LIN {X 0,Y 310.656,Z 1014.601,A -85,B 0,C 180,E1 26309.689,E2 26309.689} C_VEL
LIN {X 0,Y 289.727,Z 1045.579,A -85,B 0,C 180,E1 26313.885,E2 26313.885} C_VEL
LIN {X 0,Y 277.793,Z 1061.064,A -85,B 0,C 180,E1 26316.691,E2 26316.691} C_VEL
LIN {X 0,Y 266.703,Z 1071.977,A -85,B 0,C 180,E1 26318.403,E2 26318.403} C_VEL
LIN {X 0,Y 255.321,Z 1081.969,A -85,B 0,C 180,E1 26320.351,E2 26320.351} C_VEL
LIN {X 0,Y 233.204,Z 1105.025,A -85,B 0,C 180,E1 26328.775,E2 26328.775} C_VEL
LIN {X 0,Y 215.813,Z 1122.452,A -85,B 0,C 180,E1 26339.407,E2 26339.407} C_VEL
LIN {X 0,Y 205.814,Z 1133.022,A -85,B 0,C 180,E1 26350.657,E2 26350.657} C_VEL
LIN {X 0,Y 201.917,Z 1138.235,A -85,B 0,C 180,E1 26361.372,E2 26361.372} C_VEL
LIN {X 0,Y 201.653,Z 1139.483,A -85,B 0,C 180,E1 26370.004,E2 26370.004} C_VEL
LIN {X 0,Y 201.955,Z 1138.196,A -85,B 0,C 180,E1 26378.634,E2 26378.634} C_VEL
LIN {X 0,Y 205.859,Z 1132.908,A -85,B 0,C 180,E1 26389.346,E2 26389.346} C_VEL
LIN {X 0,Y 215.912,Z 1122.258,A -85,B 0,C 180,E1 26400.586,E2 26400.586} C_VEL
LIN {X 0,Y 233.437,Z 1104.704,A -85,B 0,C 180,E1 26411.215,E2 26411.215} C_VEL
LIN {X 0,Y 255.523,Z 1081.509,A -85,B 0,C 180,E1 26419.657,E2 26419.657} C_VEL
LIN {X 0,Y 278.933,Z 1053.943,A -85,B 0,C 180,E1 26425.937,E2 26425.937} C_VEL
LIN {X 0,Y 303.43,Z 1019.934,A -85,B 0,C 180,E1 26430.914,E2 26430.914} C_VEL
LIN {X 0,Y 325.476,Z 982.197,A -85,B 0,C 180,E1 26434.492,E2 26434.492} C_VEL
LIN {X 0,Y 325.74,Z 970.343,A -85,B 0,C 180,E1 26437.786,E2 26437.786} C_VEL
LIN {X 0,Y 324.423,Z 954.359,A -85,B 0,C 180,E1 26443.718,E2 26443.718} C_VEL
LIN {X 0,Y 322.918,Z 944.433,A -85,B 0,C 180,E1 26449.173,E2 26449.173} C_VEL
LIN {X 0,Y 322.497,Z 936.41,A -85,B 0,C 180,E1 26457.297,E2 26457.297} C_VEL
LIN {X 0,Y 322.512,Z 936.483,A -85,B 0,C 180,E1 26459.99,E2 26459.99} C_VEL
LIN {X 0,Y 322.75,Z 943.035,A -85,B 0,C 180,E1 26466.729,E2 26466.729} C_VEL
LIN {X 0,Y 324.195,Z 953.745,A -85,B 0,C 180,E1 26472.815,E2 26472.815} C_VEL
LIN {X 0,Y 325.518,Z 969.409,A -85,B 0,C 180,E1 26478.651,E2 26478.651} C_VEL
LIN {X 0,Y 325.37,Z 982.593,A -85,B 0,C 180,E1 26482.362,E2 26482.362} C_VEL
LIN {X 0,Y 303.394,Z 1021.107,A -85,B 0,C 180,E1 26485.977,E2 26485.977} C_VEL
LIN {X 0,Y 280.23,Z 1054.421,A -85,B 0,C 180,E1 26490.68,E2 26490.68} C_VEL
LIN {X 0,Y 257.476,Z 1082.65,A -85,B 0,C 180,E1 26496.694,E2 26496.694} C_VEL
LIN {X 0,Y 237.226,Z 1105.526,A -85,B 0,C 180,E1 26504.062,E2 26504.062} C_VEL
LIN {X 0,Y 219.041,Z 1125.176,A -85,B 0,C 180,E1 26513.983,E2 26513.983} C_VEL
LIN {X 0,Y 206.829,Z 1139.423,A -85,B 0,C 180,E1 26525.882,E2 26525.882} C_VEL
LIN {X 0,Y 202.177,Z 1146.947,A -85,B 0,C 180,E1 26537.003,E2 26537.003} C_VEL
LIN {X 0,Y 201.199,Z 1149.691,A -85,B 0,C 180,E1 26545.677,E2 26545.677} C_VEL
LIN {X 0,Y 201.527,Z 1150.057,A -85,B 0,C 180,E1 26549.996,E2 26549.996} C_VEL
LIN {X 0,Y 201.398,Z 1148.668,A -85,B 0,C 180,E1 26558.65,E2 26558.65} C_VEL
LIN {X 0,Y 204.311,Z 1143.178,A -85,B 0,C 180,E1 26569.491,E2 26569.491} C_VEL
LIN {X 0,Y 213.682,Z 1131.328,A -85,B 0,C 180,E1 26581.729,E2 26581.729} C_VEL
LIN {X 0,Y 229.673,Z 1113.75,A -85,B 0,C 180,E1 26592.392,E2 26592.392} C_VEL
LIN {X 0,Y 250.76,Z 1090.55,A -85,B 0,C 180,E1 26601.146,E2 26601.146} C_VEL
LIN {X 0,Y 272.752,Z 1064.306,A -85,B 0,C 180,E1 26607.53,E2 26607.53} C_VEL
LIN {X 0,Y 295.471,Z 1033.482,A -85,B 0,C 180,E1 26612.53,E2 26612.53} C_VEL
LIN {X 0,Y 318.003,Z 997.074,A -85,B 0,C 180,E1 26616.452,E2 26616.452} C_VEL
LIN {X 0,Y 325.814,Z 981.719,A -85,B 0,C 180,E1 26617.813,E2 26617.813} C_VEL
LIN {X 0,Y 325.351,Z 964.308,A -85,B 0,C 180,E1 26623.09,E2 26623.09} C_VEL
LIN {X 0,Y 324,Z 951.083,A -85,B 0,C 180,E1 26628.548,E2 26628.548} C_VEL
LIN {X 0,Y 322.759,Z 941.668,A -85,B 0,C 180,E1 26634.623,E2 26634.623} C_VEL
LIN {X 0,Y 322.742,Z 936.78,A -85,B 0,C 180,E1 26640.01,E2 26640.01} C_VEL
LIN {X 0,Y 322.687,Z 936.823,A -85,B 0,C 180,E1 26642.701,E2 26642.701} C_VEL
LIN {X 0,Y 323.156,Z 944.767,A -85,B 0,C 180,E1 26650.819,E2 26650.819} C_VEL
LIN {X 0,Y 324.807,Z 956.324,A -85,B 0,C 180,E1 26656.96,E2 26656.96} C_VEL
LIN {X 0,Y 326.013,Z 972.408,A -85,B 0,C 180,E1 26662.739,E2 26662.739} C_VEL
LIN {X 0,Y 326.137,Z 981.075,A -85,B 0,C 180,E1 26665.251,E2 26665.251} C_VEL
LIN {X 0,Y 303.951,Z 1019.446,A -85,B 0,C 180,E1 26668.904,E2 26668.904} C_VEL
LIN {X 0,Y 280.08,Z 1052.757,A -85,B 0,C 180,E1 26673.726,E2 26673.726} C_VEL
LIN {X 0,Y 255.321,Z 1081.969,A -85,B 0,C 180,E1 26680.351,E2 26680.351} C_VEL
LIN {X 0,Y 243.945,Z 1091.297,A -85,B 0,C 180,E1 26682.559,E2 26682.559} C_VEL
LIN {X 0,Y 232.748,Z 1099.829,A -85,B 0,C 180,E1 26685.058,E2 26685.058} C_VEL
LIN {X 0,Y 214.056,Z 1117.775,A -85,B 0,C 180,E1 26694.59,E2 26694.59} C_VEL
LIN {X 0,Y 201.342,Z 1130.014,A -85,B 0,C 180,E1 26705.583,E2 26705.583} C_VEL
LIN {X 0,Y 195.265,Z 1136.858,A -85,B 0,C 180,E1 26716.543,E2 26716.543} C_VEL
LIN {X 0,Y 193.614,Z 1139.385,A -85,B 0,C 180,E1 26725.516,E2 26725.516} C_VEL
LIN {X 0,Y 193.779,Z 1139.69,A -85,B 0,C 180,E1 26730.004,E2 26730.004} C_VEL
LIN {X 0,Y 194.118,Z 1138.404,A -85,B 0,C 180,E1 26738.985,E2 26738.985} C_VEL
LIN {X 0,Y 198.32,Z 1133.12,A -85,B 0,C 180,E1 26750.113,E2 26750.113} C_VEL
LIN {X 0,Y 209.02,Z 1122.475,A -85,B 0,C 180,E1 26761.709,E2 26761.709} C_VEL
LIN {X 0,Y 227.721,Z 1104.651,A -85,B 0,C 180,E1 26772.674,E2 26772.674} C_VEL
LIN {X 0,Y 250.602,Z 1081.533,A -85,B 0,C 180,E1 26781.113,E2 26781.113} C_VEL
LIN {X 0,Y 275.896,Z 1052.531,A -85,B 0,C 180,E1 26787.609,E2 26787.609} C_VEL
LIN {X 0,Y 300.384,Z 1019.113,A -85,B 0,C 180,E1 26792.364,E2 26792.364} C_VEL
LIN {X 0,Y 320.943,Z 984.275,A -85,B 0,C 180,E1 26795.727,E2 26795.727} C_VEL
LIN {X 0,Y 320.748,Z 967.42,A -85,B 0,C 180,E1 26801.325,E2 26801.325} C_VEL
LIN {X 0,Y 319.765,Z 955.09,A -85,B 0,C 180,E1 26806.984,E2 26806.984} C_VEL
LIN {X 0,Y 318.752,Z 947.169,A -85,B 0,C 180,E1 26813.041,E2 26813.041} C_VEL
LIN {X 0,Y 319.14,Z 943.671,A -85,B 0,C 180,E1 26817.269,E2 26817.269} C_VEL
LIN {X 0,Y 319.16,Z 943.724,A -85,B 0,C 180,E1 26819.99,E2 26819.99} C_VEL
LIN {X 0,Y 319.148,Z 950.325,A -85,B 0,C 180,E1 26826.806,E2 26826.806} C_VEL
LIN {X 0,Y 320.193,Z 961.352,A -85,B 0,C 180,E1 26832.978,E2 26832.978} C_VEL
LIN {X 0,Y 320.821,Z 974.906,A -85,B 0,C 180,E1 26838.092,E2 26838.092} C_VEL
LIN {X 0,Y 320.66,Z 985.105,A -85,B 0,C 180,E1 26841.15,E2 26841.15} C_VEL
LIN {X 0,Y 297.827,Z 1024.077,A -85,B 0,C 180,E1 26844.959,E2 26844.959} C_VEL
LIN {X 0,Y 272.881,Z 1058.44,A -85,B 0,C 180,E1 26849.965,E2 26849.965} C_VEL
LIN {X 0,Y 247.91,Z 1087.811,A -85,B 0,C 180,E1 26856.658,E2 26856.658} C_VEL
LIN {X 0,Y 225.003,Z 1112.055,A -85,B 0,C 180,E1 26865.528,E2 26865.528} C_VEL
LIN {X 0,Y 208.116,Z 1129.468,A -85,B 0,C 180,E1 26875.905,E2 26875.905} C_VEL
LIN {X 0,Y 197.83,Z 1141.286,A -85,B 0,C 180,E1 26887.48,E2 26887.48} C_VEL
LIN {X 0,Y 194.384,Z 1146.736,A -85,B 0,C 180,E1 26896.473,E2 26896.473} C_VEL
LIN {X 0,Y 193.286,Z 1149.483,A -85,B 0,C 180,E1 26905.5,E2 26905.5} C_VEL
LIN {X 0,Y 193.627,Z 1149.85,A -85,B 0,C 180,E1 26909.996,E2 26909.996} C_VEL
LIN {X 0,Y 193.516,Z 1148.459,A -85,B 0,C 180,E1 26919.005,E2 26919.005} C_VEL
LIN {X 0,Y 196.695,Z 1142.965,A -85,B 0,C 180,E1 26930.278,E2 26930.278} C_VEL
LIN {X 0,Y 206.766,Z 1131.11,A -85,B 0,C 180,E1 26942.922,E2 26942.922} C_VEL
LIN {X 0,Y 225.038,Z 1112.176,A -85,B 0,C 180,E1 26954.462,E2 26954.462} C_VEL
LIN {X 0,Y 247.896,Z 1087.996,A -85,B 0,C 180,E1 26963.337,E2 26963.337} C_VEL
LIN {X 0,Y 272.926,Z 1058.613,A -85,B 0,C 180,E1 26970.041,E2 26970.041} C_VEL
LIN {X 0,Y 297.899,Z 1024.305,A -85,B 0,C 180,E1 26975.04,E2 26975.04} C_VEL
LIN {X 0,Y 320.005,Z 987.274,A -85,B 0,C 180,E1 26978.578,E2 26978.578} C_VEL
LIN {X 0,Y 320.914,Z 984.537,A -85,B 0,C 180,E1 26979.05,E2 26979.05} C_VEL
LIN {X 0,Y 320.856,Z 968.383,A -85,B 0,C 180,E1 26984.257,E2 26984.257} C_VEL
LIN {X 0,Y 319.943,Z 956.175,A -85,B 0,C 180,E1 26989.712,E2 26989.712} C_VEL
LIN {X 0,Y 319.033,Z 947.677,A -85,B 0,C 180,E1 26995.786,E2 26995.786} C_VEL
LIN {X 0,Y 319.368,Z 944.031,A -85,B 0,C 180,E1 27000.01,E2 27000.01} C_VEL
LIN {X 0,Y 319.294,Z 944.109,A -85,B 0,C 180,E1 27002.73,E2 27002.73} C_VEL
LIN {X 0,Y 319.368,Z 950.839,A -85,B 0,C 180,E1 27009.986,E2 27009.986} C_VEL
LIN {X 0,Y 320.468,Z 960.823,A -85,B 0,C 180,E1 27015.784,E2 27015.784} C_VEL
LIN {X 0,Y 321.21,Z 976.997,A -85,B 0,C 180,E1 27021.908,E2 27021.908} C_VEL
LIN {X 0,Y 320.622,Z 985.751,A -85,B 0,C 180,E1 27024.382,E2 27024.382} C_VEL
LIN {X 0,Y 299.451,Z 1020.785,A -85,B 0,C 180,E1 27027.697,E2 27027.697} C_VEL
LIN {X 0,Y 275.707,Z 1053.01,A -85,B 0,C 180,E1 27032.34,E2 27032.34} C_VEL
LIN {X 0,Y 250.422,Z 1081.958,A -85,B 0,C 180,E1 27038.881,E2 27038.881} C_VEL
LIN {X 0,Y 232.748,Z 1099.829,A -85,B 0,C 180,E1 27045.058,E2 27045.058} C_VEL
LIN {X 0,Y 221.764,Z 1107.624,A -85,B 0,C 180,E1 27047.903,E2 27047.903} C_VEL
LIN {X 0,Y 211.211,Z 1114.605,A -85,B 0,C 180,E1 27051.106,E2 27051.106} C_VEL
LIN {X 0,Y 196.097,Z 1128.332,A -85,B 0,C 180,E1 27062.385,E2 27062.385} C_VEL
LIN {X 0,Y 187.522,Z 1137.066,A -85,B 0,C 180,E1 27075.976,E2 27075.976} C_VEL
LIN {X 0,Y 185.714,Z 1139.592,A -85,B 0,C 180,E1 27085.324,E2 27085.324} C_VEL
LIN {X 0,Y 185.873,Z 1139.897,A -85,B 0,C 180,E1 27090.004,E2 27090.004} C_VEL
LIN {X 0,Y 186.27,Z 1138.613,A -85,B 0,C 180,E1 27099.367,E2 27099.367} C_VEL
LIN {X 0,Y 190.839,Z 1133.33,A -85,B 0,C 180,E1 27110.937,E2 27110.937} C_VEL
LIN {X 0,Y 202.233,Z 1122.691,A -85,B 0,C 180,E1 27122.905,E2 27122.905} C_VEL
LIN {X 0,Y 221.862,Z 1104.875,A -85,B 0,C 180,E1 27134.085,E2 27134.085} C_VEL
LIN {X 0,Y 245.883,Z 1081.522,A -85,B 0,C 180,E1 27142.633,E2 27142.633} C_VEL
LIN {X 0,Y 271.691,Z 1052.79,A -85,B 0,C 180,E1 27149.035,E2 27149.035} C_VEL
LIN {X 0,Y 296.781,Z 1019.409,A -85,B 0,C 180,E1 27153.723,E2 27153.723} C_VEL
LIN {X 0,Y 315.966,Z 987.623,A -85,B 0,C 180,E1 27156.843,E2 27156.843} C_VEL
LIN {X 0,Y 316.206,Z 971.619,A -85,B 0,C 180,E1 27162.493,E2 27162.493} C_VEL
LIN {X 0,Y 315.6,Z 960.15,A -85,B 0,C 180,E1 27168.217,E2 27168.217} C_VEL
LIN {X 0,Y 315.145,Z 953.094,A -85,B 0,C 180,E1 27174.472,E2 27174.472} C_VEL
LIN {X 0,Y 315.586,Z 950.823,A -85,B 0,C 180,E1 27177.238,E2 27177.238} C_VEL
LIN {X 0,Y 315.604,Z 950.871,A -85,B 0,C 180,E1 27179.99,E2 27179.99} C_VEL
LIN {X 0,Y 315.429,Z 957.619,A -85,B 0,C 180,E1 27186.886,E2 27186.886} C_VEL
LIN {X 0,Y 315.999,Z 967.366,A -85,B 0,C 180,E1 27192.449,E2 27192.449} C_VEL
LIN {X 0,Y 316.083,Z 981.734,A -85,B 0,C 180,E1 27197.954,E2 27197.954} C_VEL
LIN {X 0,Y 315.726,Z 988.26,A -85,B 0,C 180,E1 27199.995,E2 27199.995} C_VEL
LIN {X 0,Y 311.446,Z 996.743,A -85,B 0,C 180,E1 27200.869,E2 27200.869} C_VEL
LIN {X 0,Y 286.904,Z 1034.674,A -85,B 0,C 180,E1 27204.854,E2 27204.854} C_VEL
LIN {X 0,Y 261.02,Z 1067.638,A -85,B 0,C 180,E1 27210.287,E2 27210.287} C_VEL
LIN {X 0,Y 236.125,Z 1094.834,A -85,B 0,C 180,E1 27217.354,E2 27217.354} C_VEL
LIN {X 0,Y 214.378,Z 1116.537,A -85,B 0,C 180,E1 27226.436,E2 27226.436} C_VEL
LIN {X 0,Y 197.865,Z 1132.819,A -85,B 0,C 180,E1 27237.582,E2 27237.582} C_VEL
LIN {X 0,Y 189.098,Z 1142.697,A -85,B 0,C 180,E1 27248.861,E2 27248.861} C_VEL
LIN {X 0,Y 185.658,Z 1148.233,A -85,B 0,C 180,E1 27260.602,E2 27260.602} C_VEL
LIN {X 0,Y 185.715,Z 1149.642,A -85,B 0,C 180,E1 27269.996,E2 27269.996} C_VEL
LIN {X 0,Y 186.127,Z 1147.185,A -85,B 0,C 180,E1 27282.456,E2 27282.456} C_VEL
LIN {X 0,Y 191.281,Z 1140.142,A -85,B 0,C 180,E1 27294.826,E2 27294.826} C_VEL
LIN {X 0,Y 204.521,Z 1126.321,A -85,B 0,C 180,E1 27307.66,E2 27307.66} C_VEL
LIN {X 0,Y 224.032,Z 1107.203,A -85,B 0,C 180,E1 27318.063,E2 27318.063} C_VEL
LIN {X 0,Y 247.226,Z 1083.229,A -85,B 0,C 180,E1 27326.108,E2 27326.108} C_VEL
LIN {X 0,Y 272.003,Z 1054.516,A -85,B 0,C 180,E1 27332.2,E2 27332.2} C_VEL
LIN {X 0,Y 296.648,Z 1020.872,A -85,B 0,C 180,E1 27336.827,E2 27336.827} C_VEL
LIN {X 0,Y 315.242,Z 990.373,A -85,B 0,C 180,E1 27339.661,E2 27339.661} C_VEL
LIN {X 0,Y 316.212,Z 983.473,A -85,B 0,C 180,E1 27341.563,E2 27341.563} C_VEL
LIN {X 0,Y 316.28,Z 969.136,A -85,B 0,C 180,E1 27346.859,E2 27346.859} C_VEL
LIN {X 0,Y 315.684,Z 959.928,A -85,B 0,C 180,E1 27351.732,E2 27351.732} C_VEL
LIN {X 0,Y 315.359,Z 953.613,A -85,B 0,C 180,E1 27357.257,E2 27357.257} C_VEL
LIN {X 0,Y 315.795,Z 951.212,A -85,B 0,C 180,E1 27360.01,E2 27360.01} C_VEL
LIN {X 0,Y 315.72,Z 951.302,A -85,B 0,C 180,E1 27362.761,E2 27362.761} C_VEL
LIN {X 0,Y 315.603,Z 957.552,A -85,B 0,C 180,E1 27369.683,E2 27369.683} C_VEL
LIN {X 0,Y 316.281,Z 966.936,A -85,B 0,C 180,E1 27375.287,E2 27375.287} C_VEL
LIN {X 0,Y 316.444,Z 982.685,A -85,B 0,C 180,E1 27381.422,E2 27381.422} C_VEL
LIN {X 0,Y 315.569,Z 989.407,A -85,B 0,C 180,E1 27383.343,E2 27383.343} C_VEL
LIN {X 0,Y 294.362,Z 1023.137,A -85,B 0,C 180,E1 27386.582,E2 27386.582} C_VEL
LIN {X 0,Y 270.127,Z 1054.868,A -85,B 0,C 180,E1 27391.203,E2 27391.203} C_VEL
LIN {X 0,Y 244.652,Z 1082.994,A -85,B 0,C 180,E1 27397.663,E2 27397.663} C_VEL
LIN {X 0,Y 221.552,Z 1105.307,A -85,B 0,C 180,E1 27405.966,E2 27405.966} C_VEL
LIN {X 0,Y 211.211,Z 1114.605,A -85,B 0,C 180,E1 27411.106,E2 27411.106} C_VEL
LIN {X 0,Y 201.172,Z 1120.795,A -85,B 0,C 180,E1 27414.718,E2 27414.718} C_VEL
LIN {X 0,Y 191.732,Z 1126.166,A -85,B 0,C 180,E1 27418.74,E2 27418.74} C_VEL
LIN {X 0,Y 181.895,Z 1135.042,A -85,B 0,C 180,E1 27430.542,E2 27430.542} C_VEL
LIN {X 0,Y 178.397,Z 1138.858,A -85,B 0,C 180,E1 27440.224,E2 27440.224} C_VEL
LIN {X 0,Y 177.967,Z 1140.104,A -85,B 0,C 180,E1 27450.004,E2 27450.004} C_VEL
LIN {X 0,Y 178.431,Z 1138.821,A -85,B 0,C 180,E1 27459.782,E2 27459.782} C_VEL
LIN {X 0,Y 183.396,Z 1133.542,A -85,B 0,C 180,E1 27471.83,E2 27471.83} C_VEL
LIN {X 0,Y 195.521,Z 1122.908,A -85,B 0,C 180,E1 27484.187,E2 27484.187} C_VEL
LIN {X 0,Y 215.598,Z 1105.61,A -85,B 0,C 180,E1 27495.334,E2 27495.334} C_VEL
LIN {X 0,Y 240.306,Z 1082.573,A -85,B 0,C 180,E1 27503.919,E2 27503.919} C_VEL
LIN {X 0,Y 267.655,Z 1053.048,A -85,B 0,C 180,E1 27510.506,E2 27510.506} C_VEL
LIN {X 0,Y 293.342,Z 1019.701,A -85,B 0,C 180,E1 27515.118,E2 27515.118} C_VEL
LIN {X 0,Y 311.02,Z 991.738,A -85,B 0,C 180,E1 27517.766,E2 27517.766} C_VEL
LIN {X 0,Y 311.679,Z 977.397,A -85,B 0,C 180,E1 27523.032,E2 27523.032} C_VEL
LIN {X 0,Y 311.561,Z 966.366,A -85,B 0,C 180,E1 27528.773,E2 27528.773} C_VEL
LIN {X 0,Y 311.557,Z 959.011,A -85,B 0,C 180,E1 27535.807,E2 27535.807} C_VEL
LIN {X 0,Y 311.897,Z 957.937,A -85,B 0,C 180,E1 27537.205,E2 27537.205} C_VEL
LIN {X 0,Y 311.923,Z 957.969,A -85,B 0,C 180,E1 27539.99,E2 27539.99} C_VEL
LIN {X 0,Y 311.516,Z 965.778,A -85,B 0,C 180,E1 27547.675,E2 27547.675} C_VEL
LIN {X 0,Y 311.614,Z 976.784,A -85,B 0,C 180,E1 27553.467,E2 27553.467} C_VEL
LIN {X 0,Y 310.921,Z 991.253,A -85,B 0,C 180,E1 27558.745,E2 27558.745} C_VEL
LIN {X 0,Y 310.239,Z 993.591,A -85,B 0,C 180,E1 27559.242,E2 27559.242} C_VEL
LIN {X 0,Y 287.46,Z 1028.955,A -85,B 0,C 180,E1 27562.714,E2 27562.714} C_VEL
LIN {X 0,Y 262.378,Z 1061.082,A -85,B 0,C 180,E1 27567.498,E2 27567.498} C_VEL
LIN {X 0,Y 237.267,Z 1088.591,A -85,B 0,C 180,E1 27573.879,E2 27573.879} C_VEL
LIN {X 0,Y 212.845,Z 1112.347,A -85,B 0,C 180,E1 27582.797,E2 27582.797} C_VEL
LIN {X 0,Y 193.685,Z 1130.122,A -85,B 0,C 180,E1 27594.071,E2 27594.071} C_VEL
LIN {X 0,Y 182.956,Z 1140.891,A -85,B 0,C 180,E1 27605.585,E2 27605.585} C_VEL
LIN {X 0,Y 178.8,Z 1146.315,A -85,B 0,C 180,E1 27615.268,E2 27615.268} C_VEL
LIN {X 0,Y 177.465,Z 1149.067,A -85,B 0,C 180,E1 27625.098,E2 27625.098} C_VEL
LIN {X 0,Y 177.803,Z 1149.435,A -85,B 0,C 180,E1 27629.996,E2 27629.996} C_VEL
LIN {X 0,Y 177.796,Z 1148.042,A -85,B 0,C 180,E1 27639.809,E2 27639.809} C_VEL
LIN {X 0,Y 181.618,Z 1142.54,A -85,B 0,C 180,E1 27652.045,E2 27652.045} C_VEL
LIN {X 0,Y 191.742,Z 1132.066,A -85,B 0,C 180,E1 27664.294,E2 27664.294} C_VEL
LIN {X 0,Y 208.527,Z 1116.439,A -85,B 0,C 180,E1 27675.103,E2 27675.103} C_VEL
LIN {X 0,Y 231.256,Z 1094.74,A -85,B 0,C 180,E1 27684.269,E2 27684.269} C_VEL
LIN {X 0,Y 256.981,Z 1067.632,A -85,B 0,C 180,E1 27691.28,E2 27691.28} C_VEL
LIN {X 0,Y 283.394,Z 1035.022,A -85,B 0,C 180,E1 27696.572,E2 27696.572} C_VEL
LIN {X 0,Y 308.102,Z 997.876,A -85,B 0,C 180,E1 27700.415,E2 27700.415} C_VEL
LIN {X 0,Y 310.961,Z 992.599,A -85,B 0,C 180,E1 27700.908,E2 27700.908} C_VEL
LIN {X 0,Y 311.833,Z 977.375,A -85,B 0,C 180,E1 27706.345,E2 27706.345} C_VEL
LIN {X 0,Y 311.715,Z 967.154,A -85,B 0,C 180,E1 27711.626,E2 27711.626} C_VEL
LIN {X 0,Y 311.565,Z 960.649,A -85,B 0,C 180,E1 27717.223,E2 27717.223} C_VEL
LIN {X 0,Y 312.093,Z 958.314,A -85,B 0,C 180,E1 27720.01,E2 27720.01} C_VEL
LIN {X 0,Y 312.003,Z 958.418,A -85,B 0,C 180,E1 27722.794,E2 27722.794} C_VEL
LIN {X 0,Y 311.706,Z 965.566,A -85,B 0,C 180,E1 27730.415,E2 27730.415} C_VEL
LIN {X 0,Y 311.925,Z 974.452,A -85,B 0,C 180,E1 27735.506,E2 27735.506} C_VEL
LIN {X 0,Y 311.394,Z 989.802,A -85,B 0,C 180,E1 27741.474,E2 27741.474} C_VEL
LIN {X 0,Y 310.959,Z 992.46,A -85,B 0,C 180,E1 27742.22,E2 27742.22} C_VEL
LIN {X 0,Y 288.619,Z 1026.55,A -85,B 0,C 180,E1 27745.553,E2 27745.553} C_VEL
LIN {X 0,Y 264.662,Z 1056.691,A -85,B 0,C 180,E1 27750.021,E2 27750.021} C_VEL
LIN {X 0,Y 239.497,Z 1083.532,A -85,B 0,C 180,E1 27756.238,E2 27756.238} C_VEL
LIN {X 0,Y 215.084,Z 1106.173,A -85,B 0,C 180,E1 27764.801,E2 27764.801} C_VEL
LIN {X 0,Y 195.394,Z 1123.094,A -85,B 0,C 180,E1 27775.797,E2 27775.797} C_VEL
LIN {X 0,Y 191.732,Z 1126.166,A -85,B 0,C 180,E1 27778.74,E2 27778.74} C_VEL
LIN {X 0,Y 183.089,Z 1130.708,A -85,B 0,C 180,E1 27783.194,E2 27783.194} C_VEL
LIN {X 0,Y 175.322,Z 1134.373,A -85,B 0,C 180,E1 27788.104,E2 27788.104} C_VEL
LIN {X 0,Y 170.566,Z 1139.066,A -85,B 0,C 180,E1 27799.771,E2 27799.771} C_VEL
LIN {X 0,Y 170.061,Z 1140.312,A -85,B 0,C 180,E1 27810.004,E2 27810.004} C_VEL
LIN {X 0,Y 171.466,Z 1138.008,A -85,B 0,C 180,E1 27823.528,E2 27823.528} C_VEL
LIN {X 0,Y 178.995,Z 1131.203,A -85,B 0,C 180,E1 27836.715,E2 27836.715} C_VEL
LIN {X 0,Y 195.426,Z 1117.847,A -85,B 0,C 180,E1 27849.769,E2 27849.769} C_VEL
LIN {X 0,Y 218.973,Z 1098.064,A -85,B 0,C 180,E1 27860.34,E2 27860.34} C_VEL
LIN {X 0,Y 245.525,Z 1073.017,A -85,B 0,C 180,E1 27868.057,E2 27868.057} C_VEL
LIN {X 0,Y 272.444,Z 1043.073,A -85,B 0,C 180,E1 27873.651,E2 27873.651} C_VEL
LIN {X 0,Y 298.532,Z 1007.549,A -85,B 0,C 180,E1 27877.807,E2 27877.807} C_VEL
LIN {X 0,Y 305.918,Z 995.852,A -85,B 0,C 180,E1 27878.82,E2 27878.82} C_VEL
LIN {X 0,Y 307.133,Z 983.316,A -85,B 0,C 180,E1 27883.512,E2 27883.512} C_VEL
LIN {X 0,Y 307.376,Z 973.547,A -85,B 0,C 180,E1 27888.619,E2 27888.619} C_VEL
LIN {X 0,Y 307.63,Z 966.216,A -85,B 0,C 180,E1 27895.502,E2 27895.502} C_VEL
LIN {X 0,Y 308.014,Z 964.935,A -85,B 0,C 180,E1 27897.17,E2 27897.17} C_VEL
LIN {X 0,Y 308.036,Z 964.965,A -85,B 0,C 180,E1 27899.989,E2 27899.989} C_VEL
LIN {X 0,Y 307.413,Z 971.914,A -85,B 0,C 180,E1 27907.067,E2 27907.067} C_VEL
LIN {X 0,Y 307.137,Z 982.361,A -85,B 0,C 180,E1 27912.816,E2 27912.816} C_VEL
LIN {X 0,Y 306.02,Z 995.829,A -85,B 0,C 180,E1 27917.931,E2 27917.931} C_VEL
LIN {X 0,Y 282.094,Z 1031.862,A -85,B 0,C 180,E1 27921.578,E2 27921.578} C_VEL
LIN {X 0,Y 256.659,Z 1063.167,A -85,B 0,C 180,E1 27926.34,E2 27926.34} C_VEL
LIN {X 0,Y 231.517,Z 1089.582,A -85,B 0,C 180,E1 27932.578,E2 27932.578} C_VEL
LIN {X 0,Y 206.225,Z 1113.091,A -85,B 0,C 180,E1 27941.637,E2 27941.637} C_VEL
LIN {X 0,Y 185.691,Z 1131.202,A -85,B 0,C 180,E1 27953.727,E2 27953.727} C_VEL
LIN {X 0,Y 173.992,Z 1142.411,A -85,B 0,C 180,E1 27967.16,E2 27967.16} C_VEL
LIN {X 0,Y 169.949,Z 1147.815,A -85,B 0,C 180,E1 27979.724,E2 27979.724} C_VEL
LIN {X 0,Y 169.889,Z 1149.227,A -85,B 0,C 180,E1 27989.996,E2 27989.996} C_VEL
LIN {X 0,Y 170.119,Z 1147.442,A -85,B 0,C 180,E1 28001.681,E2 28001.681} C_VEL
LIN {X 0,Y 175.637,Z 1140.702,A -85,B 0,C 180,E1 28015.547,E2 28015.547} C_VEL
LIN {X 0,Y 188.672,Z 1128.629,A -85,B 0,C 180,E1 28028.485,E2 28028.485} C_VEL
LIN {X 0,Y 208.512,Z 1111.223,A -85,B 0,C 180,E1 28039.332,E2 28039.332} C_VEL
LIN {X 0,Y 234.388,Z 1086.989,A -85,B 0,C 180,E1 28048.236,E2 28048.236} C_VEL
LIN {X 0,Y 262.485,Z 1056.82,A -85,B 0,C 180,E1 28054.853,E2 28054.853} C_VEL
LIN {X 0,Y 289.104,Z 1022.613,A -85,B 0,C 180,E1 28059.515,E2 28059.515} C_VEL
LIN {X 0,Y 306.158,Z 996.098,A -85,B 0,C 180,E1 28062.059,E2 28062.059} C_VEL
LIN {X 0,Y 307.354,Z 982.51,A -85,B 0,C 180,E1 28067.194,E2 28067.194} C_VEL
LIN {X 0,Y 307.549,Z 972.235,A -85,B 0,C 180,E1 28072.937,E2 28072.937} C_VEL
LIN {X 0,Y 308.214,Z 965.3,A -85,B 0,C 180,E1 28080.011,E2 28080.011} C_VEL
LIN {X 0,Y 308.118,Z 965.424,A -85,B 0,C 180,E1 28082.829,E2 28082.829} C_VEL
LIN {X 0,Y 307.591,Z 971.822,A -85,B 0,C 180,E1 28089.891,E2 28089.891} C_VEL
LIN {X 0,Y 307.486,Z 980.405,A -85,B 0,C 180,E1 28095.002,E2 28095.002} C_VEL
LIN {X 0,Y 306.412,Z 995.403,A -85,B 0,C 180,E1 28100.999,E2 28100.999} C_VEL
LIN {X 0,Y 281.479,Z 1031.986,A -85,B 0,C 180,E1 28104.727,E2 28104.727} C_VEL
LIN {X 0,Y 255.049,Z 1063.259,A -85,B 0,C 180,E1 28109.684,E2 28109.684} C_VEL
LIN {X 0,Y 227.124,Z 1090.982,A -85,B 0,C 180,E1 28116.912,E2 28116.912} C_VEL
LIN {X 0,Y 202.675,Z 1112.036,A -85,B 0,C 180,E1 28126.285,E2 28126.285} C_VEL
LIN {X 0,Y 183.226,Z 1127.798,A -85,B 0,C 180,E1 28138.885,E2 28138.885} C_VEL
LIN {X 0,Y 175.322,Z 1134.373,A -85,B 0,C 180,E1 28148.104,E2 28148.104} C_VEL
LIN {X 0,Y 172.468,Z 1135.92,A -85,B 0,C 180,E1 28150.785,E2 28150.785} C_VEL
LIN {X 0,Y 163.042,Z 1139.06,A -85,B 0,C 180,E1 28158.357,E2 28158.357} C_VEL
LIN {X 0,Y 162.802,Z 1139.228,A -85,B 0,C 180,E1 28159.121,E2 28159.121} C_VEL
LIN {X 0,Y 162.169,Z 1140.519,A -85,B 0,C 180,E1 28170.005,E2 28170.005} C_VEL
LIN {X 0,Y 162.81,Z 1139.237,A -85,B 0,C 180,E1 28180.732,E2 28180.732} C_VEL
LIN {X 0,Y 168.624,Z 1133.965,A -85,B 0,C 180,E1 28193.855,E2 28193.855} C_VEL
LIN {X 0,Y 183.334,Z 1122.615,A -85,B 0,C 180,E1 28207.641,E2 28207.641} C_VEL
LIN {X 0,Y 205.765,Z 1105.06,A -85,B 0,C 180,E1 28219.01,E2 28219.01} C_VEL
LIN {X 0,Y 231.826,Z 1082.457,A -85,B 0,C 180,E1 28227.303,E2 28227.303} C_VEL
LIN {X 0,Y 259.757,Z 1054.016,A -85,B 0,C 180,E1 28233.495,E2 28233.495} C_VEL
LIN {X 0,Y 286.687,Z 1020.686,A -85,B 0,C 180,E1 28237.968,E2 28237.968} C_VEL
LIN {X 0,Y 301.111,Z 999.291,A -85,B 0,C 180,E1 28239.967,E2 28239.967} C_VEL
LIN {X 0,Y 302.608,Z 986.966,A -85,B 0,C 180,E1 28244.977,E2 28244.977} C_VEL
LIN {X 0,Y 303.122,Z 978.194,A -85,B 0,C 180,E1 28250.225,E2 28250.225} C_VEL
LIN {X 0,Y 304.004,Z 971.881,A -85,B 0,C 180,E1 28257.133,E2 28257.133} C_VEL
LIN {X 0,Y 303.697,Z 972.833,A -85,B 0,C 180,E1 28261.176,E2 28261.176} C_VEL
LIN {X 0,Y 303.083,Z 979.979,A -85,B 0,C 180,E1 28267.89,E2 28267.89} C_VEL
LIN {X 0,Y 302.192,Z 991.425,A -85,B 0,C 180,E1 28273.766,E2 28273.766} C_VEL
LIN {X 0,Y 300.97,Z 1000.069,A -85,B 0,C 180,E1 28276.951,E2 28276.951} C_VEL
LIN {X 0,Y 276.863,Z 1034.76,A -85,B 0,C 180,E1 28280.409,E2 28280.409} C_VEL
LIN {X 0,Y 248.118,Z 1068.457,A -85,B 0,C 180,E1 28285.739,E2 28285.739} C_VEL
LIN {X 0,Y 219.425,Z 1096.648,A -85,B 0,C 180,E1 28293.143,E2 28293.143} C_VEL
LIN {X 0,Y 195.251,Z 1117.644,A -85,B 0,C 180,E1 28302.5,E2 28302.5} C_VEL
LIN {X 0,Y 176.304,Z 1133.333,A -85,B 0,C 180,E1 28314.513,E2 28314.513} C_VEL
LIN {X 0,Y 165.295,Z 1143.503,A -85,B 0,C 180,E1 28328.486,E2 28328.486} C_VEL
LIN {X 0,Y 162.103,Z 1147.606,A -85,B 0,C 180,E1 28339.221,E2 28339.221} C_VEL
LIN {X 0,Y 161.994,Z 1149.02,A -85,B 0,C 180,E1 28349.995,E2 28349.995} C_VEL
LIN {X 0,Y 162.089,Z 1147.625,A -85,B 0,C 180,E1 28360.77,E2 28360.77} C_VEL
LIN {X 0,Y 167.315,Z 1141.48,A -85,B 0,C 180,E1 28375.156,E2 28375.156} C_VEL
LIN {X 0,Y 180.729,Z 1129.785,A -85,B 0,C 180,E1 28388.954,E2 28388.954} C_VEL
LIN {X 0,Y 202.458,Z 1111.724,A -85,B 0,C 180,E1 28400.745,E2 28400.745} C_VEL
LIN {X 0,Y 229.986,Z 1086.96,A -85,B 0,C 180,E1 28409.909,E2 28409.909} C_VEL
LIN {X 0,Y 258.653,Z 1057.144,A -85,B 0,C 180,E1 28416.382,E2 28416.382} C_VEL
LIN {X 0,Y 286.36,Z 1022.323,A -85,B 0,C 180,E1 28421.039,E2 28421.039} C_VEL
LIN {X 0,Y 300.994,Z 1000.513,A -85,B 0,C 180,E1 28423.016,E2 28423.016} C_VEL
LIN {X 0,Y 302.559,Z 989.851,A -85,B 0,C 180,E1 28426.989,E2 28426.989} C_VEL
LIN {X 0,Y 303.229,Z 980.282,A -85,B 0,C 180,E1 28432.114,E2 28432.114} C_VEL
LIN {X 0,Y 303.792,Z 973.367,A -85,B 0,C 180,E1 28438.582,E2 28438.582} C_VEL
LIN {X 0,Y 304.208,Z 972.208,A -85,B 0,C 180,E1 28440.011,E2 28440.011} C_VEL
LIN {X 0,Y 303.764,Z 973.207,A -85,B 0,C 180,E1 28444.013,E2 28444.013} C_VEL
LIN {X 0,Y 303.302,Z 978.888,A -85,B 0,C 180,E1 28450.032,E2 28450.032} C_VEL
LIN {X 0,Y 302.646,Z 988.74,A -85,B 0,C 180,E1 28455.67,E2 28455.67} C_VEL
LIN {X 0,Y 301.132,Z 999.764,A -85,B 0,C 180,E1 28459.987,E2 28459.987} C_VEL
LIN {X 0,Y 278.241,Z 1032.248,A -85,B 0,C 180,E1 28463.237,E2 28463.237} C_VEL
LIN {X 0,Y 251.191,Z 1063.502,A -85,B 0,C 180,E1 28468.102,E2 28468.102} C_VEL
LIN {X 0,Y 222.537,Z 1091.082,A -85,B 0,C 180,E1 28475.217,E2 28475.217} C_VEL
LIN {X 0,Y 196.584,Z 1112.542,A -85,B 0,C 180,E1 28484.833,E2 28484.833} C_VEL
LIN {X 0,Y 176.395,Z 1128.01,A -85,B 0,C 180,E1 28497.536,E2 28497.536} C_VEL
LIN {X 0,Y 165.515,Z 1136.628,A -85,B 0,C 180,E1 28511.318,E2 28511.318} C_VEL
LIN {X 0,Y 162.802,Z 1139.228,A -85,B 0,C 180,E1 28519.121,E2 28519.121} C_VEL
LIN {X 0,Y 159.821,Z 1140.272,A -85,B 0,C 180,E1 28523.623,E2 28523.623} C_VEL
LIN {X 0,Y 154.108,Z 1140.646,A -85,B 0,C 180,E1 28531.431,E2 28531.431} C_VEL
LIN {X 0,Y 156.775,Z 1137.842,A -85,B 0,C 180,E1 28546.859,E2 28546.859} C_VEL
LIN {X 0,Y 168.346,Z 1129.045,A -85,B 0,C 180,E1 28562.69,E2 28562.69} C_VEL
LIN {X 0,Y 187.344,Z 1115.28,A -85,B 0,C 180,E1 28575.051,E2 28575.051} C_VEL
LIN {X 0,Y 211.805,Z 1096.225,A -85,B 0,C 180,E1 28584.594,E2 28584.594} C_VEL
LIN {X 0,Y 239.261,Z 1071.678,A -85,B 0,C 180,E1 28591.739,E2 28591.739} C_VEL
LIN {X 0,Y 267.466,Z 1041.524,A -85,B 0,C 180,E1 28597.013,E2 28597.013} C_VEL
LIN {X 0,Y 294.018,Z 1006.442,A -85,B 0,C 180,E1 28600.837,E2 28600.837} C_VEL
LIN {X 0,Y 296.549,Z 1002.134,A -85,B 0,C 180,E1 28601.368,E2 28601.368} C_VEL
LIN {X 0,Y 298.294,Z 989.713,A -85,B 0,C 180,E1 28607.068,E2 28607.068} C_VEL
LIN {X 0,Y 299.008,Z 982.259,A -85,B 0,C 180,E1 28612.712,E2 28612.712} C_VEL
LIN {X 0,Y 299.8,Z 978.709,A -85,B 0,C 180,E1 28617.093,E2 28617.093} C_VEL
LIN {X 0,Y 299.511,Z 979.625,A -85,B 0,C 180,E1 28621.192,E2 28621.192} C_VEL
LIN {X 0,Y 298.725,Z 985.867,A -85,B 0,C 180,E1 28627.273,E2 28627.273} C_VEL
LIN {X 0,Y 297.616,Z 995.506,A -85,B 0,C 180,E1 28632.53,E2 28632.53} C_VEL
LIN {X 0,Y 296.025,Z 1003.877,A -85,B 0,C 180,E1 28635.803,E2 28635.803} C_VEL
LIN {X 0,Y 270.951,Z 1038.372,A -85,B 0,C 180,E1 28639.307,E2 28639.307} C_VEL
LIN {X 0,Y 243.201,Z 1069.693,A -85,B 0,C 180,E1 28644.328,E2 28644.328} C_VEL
LIN {X 0,Y 215.075,Z 1096.42,A -85,B 0,C 180,E1 28651.324,E2 28651.324} C_VEL
LIN {X 0,Y 187.717,Z 1119.129,A -85,B 0,C 180,E1 28661.696,E2 28661.696} C_VEL
LIN {X 0,Y 167.006,Z 1135.387,A -85,B 0,C 180,E1 28675.355,E2 28675.355} C_VEL
LIN {X 0,Y 156.585,Z 1144.553,A -85,B 0,C 180,E1 28690.199,E2 28690.199} C_VEL
LIN {X 0,Y 153.733,Z 1148.442,A -85,B 0,C 180,E1 28704.339,E2 28704.339} C_VEL
LIN {X 0,Y 154.078,Z 1148.813,A -85,B 0,C 180,E1 28709.995,E2 28709.995} C_VEL
LIN {X 0,Y 154.244,Z 1147.415,A -85,B 0,C 180,E1 28721.325,E2 28721.325} C_VEL
LIN {X 0,Y 159.742,Z 1141.514,A -85,B 0,C 180,E1 28735.979,E2 28735.979} C_VEL
LIN {X 0,Y 174.46,Z 1129.569,A -85,B 0,C 180,E1 28750.639,E2 28750.639} C_VEL
LIN {X 0,Y 197.544,Z 1111.363,A -85,B 0,C 180,E1 28762.649,E2 28762.649} C_VEL
LIN {X 0,Y 224.504,Z 1088.084,A -85,B 0,C 180,E1 28771.319,E2 28771.319} C_VEL
LIN {X 0,Y 253.756,Z 1058.772,A -85,B 0,C 180,E1 28777.735,E2 28777.735} C_VEL
LIN {X 0,Y 281.399,Z 1025.274,A -85,B 0,C 180,E1 28782.235,E2 28782.235} C_VEL
LIN {X 0,Y 296.177,Z 1004.109,A -85,B 0,C 180,E1 28784.188,E2 28784.188} C_VEL
LIN {X 0,Y 298.042,Z 993.897,A -85,B 0,C 180,E1 28788.279,E2 28788.279} C_VEL
LIN {X 0,Y 298.852,Z 986.177,A -85,B 0,C 180,E1 28792.73,E2 28792.73} C_VEL
LIN {X 0,Y 299.597,Z 980.178,A -85,B 0,C 180,E1 28798.562,E2 28798.562} C_VEL
LIN {X 0,Y 300.013,Z 979.017,A -85,B 0,C 180,E1 28800.011,E2 28800.011} C_VEL
LIN {X 0,Y 299.566,Z 980.038,A -85,B 0,C 180,E1 28804.069,E2 28804.069} C_VEL
LIN {X 0,Y 298.865,Z 985.917,A -85,B 0,C 180,E1 28810.231,E2 28810.231} C_VEL
LIN {X 0,Y 297.884,Z 995.202,A -85,B 0,C 180,E1 28815.496,E2 28815.496} C_VEL
LIN {X 0,Y 296.434,Z 1003.249,A -85,B 0,C 180,E1 28818.817,E2 28818.817} C_VEL
LIN {X 0,Y 273.604,Z 1034.41,A -85,B 0,C 180,E1 28821.947,E2 28821.947} C_VEL
LIN {X 0,Y 246.037,Z 1065.231,A -85,B 0,C 180,E1 28826.761,E2 28826.761} C_VEL
LIN {X 0,Y 218.003,Z 1091.306,A -85,B 0,C 180,E1 28833.492,E2 28833.492} C_VEL
LIN {X 0,Y 190.805,Z 1112.904,A -85,B 0,C 180,E1 28843.213,E2 28843.213} C_VEL
LIN {X 0,Y 169.684,Z 1128.222,A -85,B 0,C 180,E1 28856.082,E2 28856.082} C_VEL
LIN {X 0,Y 157.965,Z 1136.837,A -85,B 0,C 180,E1 28870.389,E2 28870.389} C_VEL
LIN {X 0,Y 154.174,Z 1140.422,A -85,B 0,C 180,E1 28884.365,E2 28884.365} C_VEL
LIN {X 0,Y 154.108,Z 1140.646,A -85,B 0,C 180,E1 28891.431,E2 28891.431} C_VEL
LIN {X 0,Y 151.627,Z 1140.412,A -85,B 0,C 180,E1 28896.246,E2 28896.246} C_VEL
LIN {X 0,Y 147.723,Z 1139.2,A -85,B 0,C 180,E1 28903.681,E2 28903.681} C_VEL
LIN {X 0,Y 147.888,Z 1138.937,A -85,B 0,C 180,E1 28904.527,E2 28904.527} C_VEL
LIN {X 0,Y 156.866,Z 1132.536,A -85,B 0,C 180,E1 28919.59,E2 28919.59} C_VEL
LIN {X 0,Y 175.519,Z 1119.851,A -85,B 0,C 180,E1 28933.683,E2 28933.683} C_VEL
LIN {X 0,Y 200.572,Z 1101.672,A -85,B 0,C 180,E1 28944.306,E2 28944.306} C_VEL
LIN {X 0,Y 226.964,Z 1079.812,A -85,B 0,C 180,E1 28951.573,E2 28951.573} C_VEL
LIN {X 0,Y 255.247,Z 1052.061,A -85,B 0,C 180,E1 28957.123,E2 28957.123} C_VEL
LIN {X 0,Y 282.75,Z 1019.032,A -85,B 0,C 180,E1 28961.189,E2 28961.189} C_VEL
LIN {X 0,Y 291.345,Z 1006.998,A -85,B 0,C 180,E1 28962.293,E2 28962.293} C_VEL
LIN {X 0,Y 293.479,Z 996.853,A -85,B 0,C 180,E1 28966.852,E2 28966.852} C_VEL
LIN {X 0,Y 294.399,Z 989.563,A -85,B 0,C 180,E1 28972.056,E2 28972.056} C_VEL
LIN {X 0,Y 295.482,Z 985.46,A -85,B 0,C 180,E1 28977.05,E2 28977.05} C_VEL
LIN {X 0,Y 295.553,Z 985.415,A -85,B 0,C 180,E1 28979.989,E2 28979.989} C_VEL
LIN {X 0,Y 294.2,Z 991.833,A -85,B 0,C 180,E1 28986.736,E2 28986.736} C_VEL
LIN {X 0,Y 292.764,Z 1000.954,A -85,B 0,C 180,E1 28991.935,E2 28991.935} C_VEL
LIN {X 0,Y 291.364,Z 1007.441,A -85,B 0,C 180,E1 28994.596,E2 28994.596} C_VEL
LIN {X 0,Y 265.748,Z 1041.253,A -85,B 0,C 180,E1 28998.07,E2 28998.07} C_VEL
LIN {X 0,Y 237.714,Z 1071.635,A -85,B 0,C 180,E1 29003.005,E2 29003.005} C_VEL
LIN {X 0,Y 209.571,Z 1097.296,A -85,B 0,C 180,E1 29009.815,E2 29009.815} C_VEL
LIN {X 0,Y 182.35,Z 1118.911,A -85,B 0,C 180,E1 29019.77,E2 29019.77} C_VEL
LIN {X 0,Y 160.368,Z 1135.172,A -85,B 0,C 180,E1 29033.699,E2 29033.699} C_VEL
LIN {X 0,Y 149.009,Z 1144.341,A -85,B 0,C 180,E1 29049.147,E2 29049.147} C_VEL
LIN {X 0,Y 145.845,Z 1148.234,A -85,B 0,C 180,E1 29064.032,E2 29064.032} C_VEL
LIN {X 0,Y 146.182,Z 1148.606,A -85,B 0,C 180,E1 29069.995,E2 29069.995} C_VEL
LIN {X 0,Y 146.411,Z 1147.206,A -85,B 0,C 180,E1 29081.94,E2 29081.94} C_VEL
LIN {X 0,Y 151.665,Z 1142.039,A -85,B 0,C 180,E1 29096.018,E2 29096.018} C_VEL
LIN {X 0,Y 166.59,Z 1130.643,A -85,B 0,C 180,E1 29111.248,E2 29111.248} C_VEL
LIN {X 0,Y 189.194,Z 1113.778,A -85,B 0,C 180,E1 29123.205,E2 29123.205} C_VEL
LIN {X 0,Y 215.036,Z 1092.749,A -85,B 0,C 180,E1 29131.727,E2 29131.727} C_VEL
LIN {X 0,Y 243.189,Z 1066.454,A -85,B 0,C 180,E1 29138.065,E2 29138.065} C_VEL
LIN {X 0,Y 272.463,Z 1033.502,A -85,B 0,C 180,E1 29142.891,E2 29142.891} C_VEL
LIN {X 0,Y 291.522,Z 1007.655,A -85,B 0,C 180,E1 29145.403,E2 29145.403} C_VEL
LIN {X 0,Y 293.578,Z 997.989,A -85,B 0,C 180,E1 29149.604,E2 29149.604} C_VEL
LIN {X 0,Y 294.731,Z 989.372,A -85,B 0,C 180,E1 29155.589,E2 29155.589} C_VEL
LIN {X 0,Y 295.69,Z 985.755,A -85,B 0,C 180,E1 29160.011,E2 29160.011} C_VEL
LIN {X 0,Y 295.122,Z 986.958,A -85,B 0,C 180,E1 29164.427,E2 29164.427} C_VEL
LIN {X 0,Y 294.255,Z 992.799,A -85,B 0,C 180,E1 29170.394,E2 29170.394} C_VEL
LIN {X 0,Y 292.663,Z 1002.346,A -85,B 0,C 180,E1 29175.706,E2 29175.706} C_VEL
LIN {X 0,Y 291.418,Z 1007.357,A -85,B 0,C 180,E1 29177.637,E2 29177.637} C_VEL
LIN {X 0,Y 264.332,Z 1042.27,A -85,B 0,C 180,E1 29181.345,E2 29181.345} C_VEL
LIN {X 0,Y 235.115,Z 1072.597,A -85,B 0,C 180,E1 29186.553,E2 29186.553} C_VEL
LIN {X 0,Y 206.342,Z 1097.357,A -85,B 0,C 180,E1 29193.787,E2 29193.787} C_VEL
LIN {X 0,Y 181.593,Z 1115.7,A -85,B 0,C 180,E1 29203.114,E2 29203.114} C_VEL
LIN {X 0,Y 161.564,Z 1129.385,A -85,B 0,C 180,E1 29215.764,E2 29215.764} C_VEL
LIN {X 0,Y 149.121,Z 1138.11,A -85,B 0,C 180,E1 29232.258,E2 29232.258} C_VEL
LIN {X 0,Y 146.284,Z 1140.63,A -85,B 0,C 180,E1 29244.06,E2 29244.06} C_VEL
LIN {X 0,Y 146.223,Z 1140.862,A -85,B 0,C 180,E1 29251.34,E2 29251.34} C_VEL
LIN {X 0,Y 147.888,Z 1138.937,A -85,B 0,C 180,E1 29264.527,E2 29264.527} C_VEL
LIN {X 0,Y 147.38,Z 1137.591,A -85,B 0,C 180,E1 29269.593,E2 29269.593} C_VEL
LIN {X 0,Y 146.721,Z 1134.802,A -85,B 0,C 180,E1 29277.26,E2 29277.26} C_VEL
LIN {X 0,Y 147.266,Z 1134.378,A -85,B 0,C 180,E1 29278.076,E2 29278.076} C_VEL
LIN {X 0,Y 164.269,Z 1123.659,A -85,B 0,C 180,E1 29292.424,E2 29292.424} C_VEL
LIN {X 0,Y 190.782,Z 1105.729,A -85,B 0,C 180,E1 29304.499,E2 29304.499} C_VEL
LIN {X 0,Y 219.739,Z 1083.157,A -85,B 0,C 180,E1 29312.601,E2 29312.601} C_VEL
LIN {X 0,Y 250.567,Z 1054.147,A -85,B 0,C 180,E1 29318.523,E2 29318.523} C_VEL
LIN {X 0,Y 279.475,Z 1020.427,A -85,B 0,C 180,E1 29322.628,E2 29322.628} C_VEL
LIN {X 0,Y 286.444,Z 1010.901,A -85,B 0,C 180,E1 29323.49,E2 29323.49} C_VEL
LIN {X 0,Y 288.817,Z 1001.642,A -85,B 0,C 180,E1 29327.876,E2 29327.876} C_VEL
LIN {X 0,Y 290.189,Z 994.368,A -85,B 0,C 180,E1 29333.995,E2 29333.995} C_VEL
LIN {X 0,Y 290.986,Z 992.075,A -85,B 0,C 180,E1 29337.004,E2 29337.004} C_VEL
LIN {X 0,Y 291.05,Z 992.032,A -85,B 0,C 180,E1 29339.989,E2 29339.989} C_VEL
LIN {X 0,Y 289.637,Z 997.879,A -85,B 0,C 180,E1 29346.29,E2 29346.29} C_VEL
LIN {X 0,Y 287.561,Z 1008.065,A -85,B 0,C 180,E1 29352.154,E2 29352.154} C_VEL
LIN {X 0,Y 287.038,Z 1010.414,A -85,B 0,C 180,E1 29353.189,E2 29353.189} C_VEL
LIN {X 0,Y 259.353,Z 1045.679,A -85,B 0,C 180,E1 29356.969,E2 29356.969} C_VEL
LIN {X 0,Y 227.754,Z 1077.982,A -85,B 0,C 180,E1 29362.56,E2 29362.56} C_VEL
LIN {X 0,Y 197.5,Z 1103.578,A -85,B 0,C 180,E1 29370.206,E2 29370.206} C_VEL
LIN {X 0,Y 170.529,Z 1123.401,A -85,B 0,C 180,E1 29380.948,E2 29380.948} C_VEL
LIN {X 0,Y 152.256,Z 1136.012,A -85,B 0,C 180,E1 29393.333,E2 29393.333} C_VEL
LIN {X 0,Y 141.487,Z 1144.128,A -85,B 0,C 180,E1 29407.982,E2 29407.982} C_VEL
LIN {X 0,Y 137.939,Z 1148.026,A -85,B 0,C 180,E1 29423.688,E2 29423.688} C_VEL
LIN {X 0,Y 138.263,Z 1148.398,A -85,B 0,C 180,E1 29429.995,E2 29429.995} C_VEL
LIN {X 0,Y 138.607,Z 1146.997,A -85,B 0,C 180,E1 29442.623,E2 29442.623} C_VEL
LIN {X 0,Y 144.415,Z 1141.826,A -85,B 0,C 180,E1 29457.431,E2 29457.431} C_VEL
LIN {X 0,Y 160.553,Z 1130.429,A -85,B 0,C 180,E1 29473.166,E2 29473.166} C_VEL
LIN {X 0,Y 184.407,Z 1113.557,A -85,B 0,C 180,E1 29485.242,E2 29485.242} C_VEL
LIN {X 0,Y 211.302,Z 1092.519,A -85,B 0,C 180,E1 29493.671,E2 29493.671} C_VEL
LIN {X 0,Y 240.266,Z 1066.206,A -85,B 0,C 180,E1 29499.866,E2 29499.866} C_VEL
LIN {X 0,Y 269.363,Z 1034.284,A -85,B 0,C 180,E1 29504.414,E2 29504.414} C_VEL
LIN {X 0,Y 287.232,Z 1010.548,A -85,B 0,C 180,E1 29506.825,E2 29506.825} C_VEL
LIN {X 0,Y 289.238,Z 1000.935,A -85,B 0,C 180,E1 29511.73,E2 29511.73} C_VEL
LIN {X 0,Y 290.429,Z 994.679,A -85,B 0,C 180,E1 29517.021,E2 29517.021} C_VEL
LIN {X 0,Y 291.186,Z 992.373,A -85,B 0,C 180,E1 29520.011,E2 29520.011} C_VEL
LIN {X 0,Y 290.626,Z 993.585,A -85,B 0,C 180,E1 29524.496,E2 29524.496} C_VEL
LIN {X 0,Y 289.423,Z 999.633,A -85,B 0,C 180,E1 29530.57,E2 29530.57} C_VEL
LIN {X 0,Y 287.187,Z 1010.063,A -85,B 0,C 180,E1 29536.193,E2 29536.193} C_VEL
LIN {X 0,Y 259.907,Z 1044.357,A -85,B 0,C 180,E1 29539.952,E2 29539.952} C_VEL
LIN {X 0,Y 230.215,Z 1074.182,A -85,B 0,C 180,E1 29545.071,E2 29545.071} C_VEL
LIN {X 0,Y 201.125,Z 1098.259,A -85,B 0,C 180,E1 29552.148,E2 29552.148} C_VEL
LIN {X 0,Y 173.962,Z 1117.418,A -85,B 0,C 180,E1 29562.247,E2 29562.247} C_VEL
LIN {X 0,Y 154.975,Z 1129.597,A -85,B 0,C 180,E1 29574.089,E2 29574.089} C_VEL
LIN {X 0,Y 141.554,Z 1138.318,A -85,B 0,C 180,E1 29591.275,E2 29591.275} C_VEL
LIN {X 0,Y 138.398,Z 1140.837,A -85,B 0,C 180,E1 29603.72,E2 29603.72} C_VEL
LIN {X 0,Y 138.462,Z 1141.141,A -85,B 0,C 180,E1 29610.005,E2 29610.005} C_VEL
LIN {X 0,Y 140.072,Z 1139.253,A -85,B 0,C 180,E1 29624.925,E2 29624.925} C_VEL
LIN {X 0,Y 147.266,Z 1134.378,A -85,B 0,C 180,E1 29638.076,E2 29638.076} C_VEL
LIN {X 0,Y 149.371,Z 1131.069,A -85,B 0,C 180,E1 29644.678,E2 29644.678} C_VEL
LIN {X 0,Y 153.102,Z 1127.017,A -85,B 0,C 180,E1 29650.999,E2 29650.999} C_VEL
LIN {X 0,Y 177.782,Z 1111.639,A -85,B 0,C 180,E1 29663.491,E2 29663.491} C_VEL
LIN {X 0,Y 207.241,Z 1090.512,A -85,B 0,C 180,E1 29672.441,E2 29672.441} C_VEL
LIN {X 0,Y 237.924,Z 1064.077,A -85,B 0,C 180,E1 29678.656,E2 29678.656} C_VEL
LIN {X 0,Y 268.233,Z 1031.813,A -85,B 0,C 180,E1 29683.096,E2 29683.096} C_VEL
LIN {X 0,Y 281.556,Z 1014.859,A -85,B 0,C 180,E1 29684.714,E2 29684.714} C_VEL
LIN {X 0,Y 283.706,Z 1008.602,A -85,B 0,C 180,E1 29687.655,E2 29687.655} C_VEL
LIN {X 0,Y 285.211,Z 1001.724,A -85,B 0,C 180,E1 29692.975,E2 29692.975} C_VEL
LIN {X 0,Y 286.355,Z 998.642,A -85,B 0,C 180,E1 29696.956,E2 29696.956} C_VEL
LIN {X 0,Y 286.454,Z 998.563,A -85,B 0,C 180,E1 29699.989,E2 29699.989} C_VEL
LIN {X 0,Y 284.539,Z 1005.183,A -85,B 0,C 180,E1 29706.869,E2 29706.869} C_VEL
LIN {X 0,Y 282.517,Z 1013.313,A -85,B 0,C 180,E1 29711.531,E2 29711.531} C_VEL
LIN {X 0,Y 281.669,Z 1015.21,A -85,B 0,C 180,E1 29712.165,E2 29712.165} C_VEL
LIN {X 0,Y 254.623,Z 1048.087,A -85,B 0,C 180,E1 29715.595,E2 29715.595} C_VEL
LIN {X 0,Y 224.661,Z 1077.804,A -85,B 0,C 180,E1 29720.639,E2 29720.639} C_VEL
LIN {X 0,Y 192.425,Z 1104.154,A -85,B 0,C 180,E1 29728.434,E2 29728.434} C_VEL
LIN {X 0,Y 163.052,Z 1124.686,A -85,B 0,C 180,E1 29739.94,E2 29739.94} C_VEL
LIN {X 0,Y 142.782,Z 1137.787,A -85,B 0,C 180,E1 29754.286,E2 29754.286} C_VEL
LIN {X 0,Y 132.688,Z 1145.048,A -85,B 0,C 180,E1 29769.96,E2 29769.96} C_VEL
LIN {X 0,Y 130.041,Z 1147.817,A -85,B 0,C 180,E1 29783.303,E2 29783.303} C_VEL
LIN {X 0,Y 130.343,Z 1148.19,A -85,B 0,C 180,E1 29789.994,E2 29789.994} C_VEL
LIN {X 0,Y 130.805,Z 1146.787,A -85,B 0,C 180,E1 29803.389,E2 29803.389} C_VEL
LIN {X 0,Y 137.762,Z 1141.237,A -85,B 0,C 180,E1 29819.711,E2 29819.711} C_VEL
LIN {X 0,Y 156.391,Z 1129.092,A -85,B 0,C 180,E1 29836.338,E2 29836.338} C_VEL
LIN {X 0,Y 182.441,Z 1111.559,A -85,B 0,C 180,E1 29848.34,E2 29848.34} C_VEL
LIN {X 0,Y 213.808,Z 1087.397,A -85,B 0,C 180,E1 29857.101,E2 29857.101} C_VEL
LIN {X 0,Y 245.569,Z 1058.037,A -85,B 0,C 180,E1 29862.998,E2 29862.998} C_VEL
LIN {X 0,Y 274.982,Z 1024.419,A -85,B 0,C 180,E1 29867.066,E2 29867.066} C_VEL
LIN {X 0,Y 282.45,Z 1014.376,A -85,B 0,C 180,E1 29868.046,E2 29868.046} C_VEL
LIN {X 0,Y 284.781,Z 1005.054,A -85,B 0,C 180,E1 29873.404,E2 29873.404} C_VEL
LIN {X 0,Y 286.564,Z 998.908,A -85,B 0,C 180,E1 29880.011,E2 29880.011} C_VEL
LIN {X 0,Y 286.426,Z 999.055,A -85,B 0,C 180,E1 29883.043,E2 29883.043} C_VEL
LIN {X 0,Y 284.653,Z 1005.329,A -85,B 0,C 180,E1 29889.973,E2 29889.973} C_VEL
LIN {X 0,Y 282.369,Z 1014.051,A -85,B 0,C 180,E1 29895.025,E2 29895.025} C_VEL
LIN {X 0,Y 255.64,Z 1046.342,A -85,B 0,C 180,E1 29898.512,E2 29898.512} C_VEL
LIN {X 0,Y 225.438,Z 1075.68,A -85,B 0,C 180,E1 29903.524,E2 29903.524} C_VEL
LIN {X 0,Y 194.264,Z 1100.44,A -85,B 0,C 180,E1 29910.921,E2 29910.921} C_VEL
LIN {X 0,Y 166.381,Z 1119.132,A -85,B 0,C 180,E1 29921.304,E2 29921.304} C_VEL
LIN {X 0,Y 145.338,Z 1131.682,A -85,B 0,C 180,E1 29935.02,E2 29935.02} C_VEL
LIN {X 0,Y 134.008,Z 1138.527,A -85,B 0,C 180,E1 29950.178,E2 29950.178} C_VEL
LIN {X 0,Y 130.546,Z 1141.044,A -85,B 0,C 180,E1 29963.341,E2 29963.341} C_VEL
LIN {X 0,Y 130.552,Z 1141.348,A -85,B 0,C 180,E1 29970.006,E2 29970.006} C_VEL
LIN {X 0,Y 131.697,Z 1140.071,A -85,B 0,C 180,E1 29983.309,E2 29983.309} C_VEL
LIN {X 0,Y 141.415,Z 1133.898,A -85,B 0,C 180,E1 30000.967,E2 30000.967} C_VEL
LIN {X 0,Y 153.102,Z 1127.017,A -85,B 0,C 180,E1 30010.999,E2 30010.999} C_VEL
LIN {X 0,Y 158.286,Z 1122.354,A -85,B 0,C 180,E1 30016.925,E2 30016.925} C_VEL
LIN {X 0,Y 164.818,Z 1116.962,A -85,B 0,C 180,E1 30022.375,E2 30022.375} C_VEL
LIN {X 0,Y 193.692,Z 1098.047,A -85,B 0,C 180,E1 30031.992,E2 30031.992} C_VEL
LIN {X 0,Y 225.305,Z 1073.155,A -85,B 0,C 180,E1 30038.804,E2 30038.804} C_VEL
LIN {X 0,Y 256.701,Z 1042.589,A -85,B 0,C 180,E1 30043.577,E2 30043.577} C_VEL
LIN {X 0,Y 276.885,Z 1018.713,A -85,B 0,C 180,E1 30045.985,E2 30045.985} C_VEL
LIN {X 0,Y 279.065,Z 1012.753,A -85,B 0,C 180,E1 30049.033,E2 30049.033} C_VEL
LIN {X 0,Y 280.586,Z 1007.415,A -85,B 0,C 180,E1 30053.789,E2 30053.789} C_VEL
LIN {X 0,Y 281.553,Z 1005.065,A -85,B 0,C 180,E1 30056.904,E2 30056.904} C_VEL
LIN {X 0,Y 281.658,Z 1004.969,A -85,B 0,C 180,E1 30059.988,E2 30059.988} C_VEL
LIN {X 0,Y 279.791,Z 1010.722,A -85,B 0,C 180,E1 30066.205,E2 30066.205} C_VEL
LIN {X 0,Y 277.551,Z 1018.089,A -85,B 0,C 180,E1 30070.681,E2 30070.681} C_VEL
LIN {X 0,Y 250.043,Z 1050.462,A -85,B 0,C 180,E1 30074.166,E2 30074.166} C_VEL
LIN {X 0,Y 220.314,Z 1078.913,A -85,B 0,C 180,E1 30078.971,E2 30078.971} C_VEL
LIN {X 0,Y 188.656,Z 1103.928,A -85,B 0,C 180,E1 30086.242,E2 30086.242} C_VEL
LIN {X 0,Y 157.915,Z 1124.467,A -85,B 0,C 180,E1 30097.66,E2 30097.66} C_VEL
LIN {X 0,Y 136.12,Z 1137.658,A -85,B 0,C 180,E1 30112.419,E2 30112.419} C_VEL
LIN {X 0,Y 125.156,Z 1144.837,A -85,B 0,C 180,E1 30128.698,E2 30128.698} C_VEL
LIN {X 0,Y 122.141,Z 1147.609,A -85,B 0,C 180,E1 30142.868,E2 30142.868} C_VEL
LIN {X 0,Y 122.422,Z 1147.983,A -85,B 0,C 180,E1 30149.994,E2 30149.994} C_VEL
LIN {X 0,Y 123.04,Z 1146.578,A -85,B 0,C 180,E1 30164.252,E2 30164.252} C_VEL
LIN {X 0,Y 130.752,Z 1141.047,A -85,B 0,C 180,E1 30181.424,E2 30181.424} C_VEL
LIN {X 0,Y 150.604,Z 1129.052,A -85,B 0,C 180,E1 30198.416,E2 30198.416} C_VEL
LIN {X 0,Y 178.284,Z 1111.34,A -85,B 0,C 180,E1 30210.579,E2 30210.579} C_VEL
LIN {X 0,Y 210.768,Z 1087.169,A -85,B 0,C 180,E1 30219.144,E2 30219.144} C_VEL
LIN {X 0,Y 243.311,Z 1057.791,A -85,B 0,C 180,E1 30224.834,E2 30224.834} C_VEL
LIN {X 0,Y 273.676,Z 1023.674,A -85,B 0,C 180,E1 30228.758,E2 30228.758} C_VEL
LIN {X 0,Y 277.642,Z 1018.539,A -85,B 0,C 180,E1 30229.191,E2 30229.191} C_VEL
LIN {X 0,Y 279.933,Z 1010.965,A -85,B 0,C 180,E1 30233.798,E2 30233.798} C_VEL
LIN {X 0,Y 281.767,Z 1005.314,A -85,B 0,C 180,E1 30240.012,E2 30240.012} C_VEL
LIN {X 0,Y 281.626,Z 1005.474,A -85,B 0,C 180,E1 30243.095,E2 30243.095} C_VEL
LIN {X 0,Y 279.822,Z 1010.931,A -85,B 0,C 180,E1 30249.36,E2 30249.36} C_VEL
LIN {X 0,Y 277.877,Z 1017.299,A -85,B 0,C 180,E1 30253.41,E2 30253.41} C_VEL
LIN {X 0,Y 275.65,Z 1020.719,A -85,B 0,C 180,E1 30254.049,E2 30254.049} C_VEL
LIN {X 0,Y 245.507,Z 1054.604,A -85,B 0,C 180,E1 30257.874,E2 30257.874} C_VEL
LIN {X 0,Y 212.73,Z 1083.916,A -85,B 0,C 180,E1 30263.515,E2 30263.515} C_VEL
LIN {X 0,Y 181.784,Z 1106.414,A -85,B 0,C 180,E1 30271.322,E2 30271.322} C_VEL
LIN {X 0,Y 152.104,Z 1124.587,A -85,B 0,C 180,E1 30283.771,E2 30283.771} C_VEL
LIN {X 0,Y 132.084,Z 1135.602,A -85,B 0,C 180,E1 30300.125,E2 30300.125} C_VEL
LIN {X 0,Y 123.907,Z 1140.315,A -85,B 0,C 180,E1 30315.85,E2 30315.85} C_VEL
LIN {X 0,Y 122.643,Z 1141.555,A -85,B 0,C 180,E1 30330.006,E2 30330.006} C_VEL
LIN {X 0,Y 123.971,Z 1140.28,A -85,B 0,C 180,E1 30344.155,E2 30344.155} C_VEL
LIN {X 0,Y 132.188,Z 1135.471,A -85,B 0,C 180,E1 30359.937,E2 30359.937} C_VEL
LIN {X 0,Y 152.028,Z 1124.548,A -85,B 0,C 180,E1 30376.065,E2 30376.065} C_VEL
LIN {X 0,Y 164.818,Z 1116.962,A -85,B 0,C 180,E1 30382.375,E2 30382.375} C_VEL
LIN {X 0,Y 172.522,Z 1110.953,A -85,B 0,C 180,E1 30387.326,E2 30387.326} C_VEL
LIN {X 0,Y 181.122,Z 1104.234,A -85,B 0,C 180,E1 30391.774,E2 30391.774} C_VEL
LIN {X 0,Y 212.818,Z 1081.361,A -85,B 0,C 180,E1 30399.024,E2 30399.024} C_VEL
LIN {X 0,Y 244.75,Z 1052.937,A -85,B 0,C 180,E1 30404.054,E2 30404.054} C_VEL
LIN {X 0,Y 272.854,Z 1021.629,A -85,B 0,C 180,E1 30407.541,E2 30407.541} C_VEL
LIN {X 0,Y 275.148,Z 1014.862,A -85,B 0,C 180,E1 30412.417,E2 30412.417} C_VEL
LIN {X 0,Y 276.623,Z 1011.422,A -85,B 0,C 180,E1 30416.849,E2 30416.849} C_VEL
LIN {X 0,Y 276.758,Z 1011.306,A -85,B 0,C 180,E1 30419.988,E2 30419.988} C_VEL
LIN {X 0,Y 274.458,Z 1017.325,A -85,B 0,C 180,E1 30426.41,E2 30426.41} C_VEL
LIN {X 0,Y 273.076,Z 1021.593,A -85,B 0,C 180,E1 30429.126,E2 30429.126} C_VEL
LIN {X 0,Y 271.315,Z 1024.113,A -85,B 0,C 180,E1 30429.667,E2 30429.667} C_VEL
LIN {X 0,Y 241.324,Z 1057.252,A -85,B 0,C 180,E1 30433.288,E2 30433.288} C_VEL
LIN {X 0,Y 208.039,Z 1086.729,A -85,B 0,C 180,E1 30438.763,E2 30438.763} C_VEL
LIN {X 0,Y 174.447,Z 1110.975,A -85,B 0,C 180,E1 30447.084,E2 30447.084} C_VEL
LIN {X 0,Y 144.393,Z 1129.29,A -85,B 0,C 180,E1 30459.703,E2 30459.703} C_VEL
LIN {X 0,Y 123.887,Z 1140.769,A -85,B 0,C 180,E1 30476.601,E2 30476.601} C_VEL
LIN {X 0,Y 115.315,Z 1146.348,A -85,B 0,C 180,E1 30494.758,E2 30494.758} C_VEL
LIN {X 0,Y 114.526,Z 1147.776,A -85,B 0,C 180,E1 30509.993,E2 30509.993} C_VEL
LIN {X 0,Y 115.287,Z 1146.368,A -85,B 0,C 180,E1 30525.232,E2 30525.232} C_VEL
LIN {X 0,Y 123.889,Z 1140.835,A -85,B 0,C 180,E1 30543.384,E2 30543.384} C_VEL
LIN {X 0,Y 144.335,Z 1129.411,A -85,B 0,C 180,E1 30560.279,E2 30560.279} C_VEL
LIN {X 0,Y 174.409,Z 1111.121,A -85,B 0,C 180,E1 30572.921,E2 30572.921} C_VEL
LIN {X 0,Y 208.009,Z 1086.942,A -85,B 0,C 180,E1 30581.24,E2 30581.24} C_VEL
LIN {X 0,Y 241.31,Z 1057.546,A -85,B 0,C 180,E1 30586.699,E2 30586.699} C_VEL
LIN {X 0,Y 271.933,Z 1023.744,A -85,B 0,C 180,E1 30590.391,E2 30590.391} C_VEL
LIN {X 0,Y 273.528,Z 1020.967,A -85,B 0,C 180,E1 30591.331,E2 30591.331} C_VEL
LIN {X 0,Y 275.8,Z 1013.964,A -85,B 0,C 180,E1 30596.863,E2 30596.863} C_VEL
LIN {X 0,Y 276.86,Z 1011.629,A -85,B 0,C 180,E1 30600.012,E2 30600.012} C_VEL
LIN {X 0,Y 276.687,Z 1011.804,A -85,B 0,C 180,E1 30603.151,E2 30603.151} C_VEL
LIN {X 0,Y 274.551,Z 1017.426,A -85,B 0,C 180,E1 30609.541,E2 30609.541} C_VEL
LIN {X 0,Y 273.189,Z 1021.433,A -85,B 0,C 180,E1 30612.163,E2 30612.163} C_VEL
LIN {X 0,Y 269.826,Z 1025.773,A -85,B 0,C 180,E1 30612.852,E2 30612.852} C_VEL
LIN {X 0,Y 241.433,Z 1056.486,A -85,B 0,C 180,E1 30616.32,E2 30616.32} C_VEL
LIN {X 0,Y 209.66,Z 1084.14,A -85,B 0,C 180,E1 30621.505,E2 30621.505} C_VEL
LIN {X 0,Y 177.733,Z 1106.633,A -85,B 0,C 180,E1 30629.105,E2 30629.105} C_VEL
LIN {X 0,Y 146.645,Z 1124.8,A -85,B 0,C 180,E1 30641.497,E2 30641.497} C_VEL
LIN {X 0,Y 125.981,Z 1135.387,A -85,B 0,C 180,E1 30657.379,E2 30657.379} C_VEL
LIN {X 0,Y 116.2,Z 1140.523,A -85,B 0,C 180,E1 30674.89,E2 30674.89} C_VEL
LIN {X 0,Y 114.754,Z 1141.762,A -85,B 0,C 180,E1 30690.007,E2 30690.007} C_VEL
LIN {X 0,Y 116.262,Z 1140.488,A -85,B 0,C 180,E1 30705.115,E2 30705.115} C_VEL
LIN {X 0,Y 126.111,Z 1135.244,A -85,B 0,C 180,E1 30722.713,E2 30722.713} C_VEL
LIN {X 0,Y 146.764,Z 1124.638,A -85,B 0,C 180,E1 30738.466,E2 30738.466} C_VEL
LIN {X 0,Y 175.013,Z 1108.189,A -85,B 0,C 180,E1 30749.976,E2 30749.976} C_VEL
LIN {X 0,Y 181.122,Z 1104.234,A -85,B 0,C 180,E1 30751.774,E2 30751.774} C_VEL
LIN {X 0,Y 190.517,Z 1096.895,A -85,B 0,C 180,E1 30755.745,E2 30755.745} C_VEL
LIN {X 0,Y 200.392,Z 1088.876,A -85,B 0,C 180,E1 30759.284,E2 30759.284} C_VEL
LIN {X 0,Y 231.98,Z 1063.235,A -85,B 0,C 180,E1 30764.46,E2 30764.46} C_VEL
LIN {X 0,Y 263.156,Z 1031.608,A -85,B 0,C 180,E1 30768.196,E2 30768.196} C_VEL
LIN {X 0,Y 267.394,Z 1026.597,A -85,B 0,C 180,E1 30768.628,E2 30768.628} C_VEL
LIN {X 0,Y 268.986,Z 1023.559,A -85,B 0,C 180,E1 30770.26,E2 30770.26} C_VEL
LIN {X 0,Y 271.513,Z 1017.65,A -85,B 0,C 180,E1 30776.789,E2 30776.789} C_VEL
LIN {X 0,Y 271.674,Z 1017.493,A -85,B 0,C 180,E1 30779.988,E2 30779.988} C_VEL
LIN {X 0,Y 269.125,Z 1023.627,A -85,B 0,C 180,E1 30786.452,E2 30786.452} C_VEL
LIN {X 0,Y 268.237,Z 1025.808,A -85,B 0,C 180,E1 30787.933,E2 30787.933} C_VEL
LIN {X 0,Y 258.972,Z 1036.774,A -85,B 0,C 180,E1 30789.123,E2 30789.123} C_VEL
LIN {X 0,Y 228.43,Z 1067.414,A -85,B 0,C 180,E1 30792.91,E2 30792.91} C_VEL
LIN {X 0,Y 194.507,Z 1094.786,A -85,B 0,C 180,E1 30798.792,E2 30798.792} C_VEL
LIN {X 0,Y 160.706,Z 1116.952,A -85,B 0,C 180,E1 30807.861,E2 30807.861} C_VEL
LIN {X 0,Y 131.74,Z 1133.011,A -85,B 0,C 180,E1 30821.611,E2 30821.611} C_VEL
LIN {X 0,Y 114.499,Z 1142.014,A -85,B 0,C 180,E1 30838.033,E2 30838.033} C_VEL
LIN {X 0,Y 107.609,Z 1146.138,A -85,B 0,C 180,E1 30853.637,E2 30853.637} C_VEL
LIN {X 0,Y 106.602,Z 1147.568,A -85,B 0,C 180,E1 30869.993,E2 30869.993} C_VEL
LIN {X 0,Y 107.568,Z 1146.159,A -85,B 0,C 180,E1 30886.355,E2 30886.355} C_VEL
LIN {X 0,Y 117.196,Z 1140.621,A -85,B 0,C 180,E1 30905.568,E2 30905.568} C_VEL
LIN {X 0,Y 139.251,Z 1129.196,A -85,B 0,C 180,E1 30922.868,E2 30922.868} C_VEL
LIN {X 0,Y 170.798,Z 1110.924,A -85,B 0,C 180,E1 30935.357,E2 30935.357} C_VEL
LIN {X 0,Y 205.548,Z 1086.715,A -85,B 0,C 180,E1 30943.377,E2 30943.377} C_VEL
LIN {X 0,Y 240.653,Z 1056.263,A -85,B 0,C 180,E1 30948.736,E2 30948.736} C_VEL
LIN {X 0,Y 267.907,Z 1026.768,A -85,B 0,C 180,E1 30951.813,E2 30951.813} C_VEL
LIN {X 0,Y 270.028,Z 1021.901,A -85,B 0,C 180,E1 30955.184,E2 30955.184} C_VEL
LIN {X 0,Y 271.782,Z 1017.807,A -85,B 0,C 180,E1 30960.012,E2 30960.012} C_VEL
LIN {X 0,Y 271.581,Z 1018.026,A -85,B 0,C 180,E1 30963.21,E2 30963.21} C_VEL
LIN {X 0,Y 269.562,Z 1022.728,A -85,B 0,C 180,E1 30968.803,E2 30968.803} C_VEL
LIN {X 0,Y 267.734,Z 1026.557,A -85,B 0,C 180,E1 30971.239,E2 30971.239} C_VEL
LIN {X 0,Y 238.058,Z 1057.878,A -85,B 0,C 180,E1 30974.64,E2 30974.64} C_VEL
LIN {X 0,Y 206.857,Z 1084.363,A -85,B 0,C 180,E1 30979.44,E2 30979.44} C_VEL
LIN {X 0,Y 173.907,Z 1106.891,A -85,B 0,C 180,E1 30986.808,E2 30986.808} C_VEL
LIN {X 0,Y 141.437,Z 1125.012,A -85,B 0,C 180,E1 30999.052,E2 30999.052} C_VEL
LIN {X 0,Y 119.289,Z 1135.598,A -85,B 0,C 180,E1 31015.297,E2 31015.297} C_VEL
LIN {X 0,Y 108.537,Z 1140.731,A -85,B 0,C 180,E1 31033.795,E2 31033.795} C_VEL
LIN {X 0,Y 106.842,Z 1141.97,A -85,B 0,C 180,E1 31050.007,E2 31050.007} C_VEL
LIN {X 0,Y 108.589,Z 1140.697,A -85,B 0,C 180,E1 31066.211,E2 31066.211} C_VEL
LIN {X 0,Y 119.432,Z 1135.456,A -85,B 0,C 180,E1 31084.796,E2 31084.796} C_VEL
LIN {X 0,Y 141.547,Z 1124.854,A -85,B 0,C 180,E1 31100.91,E2 31100.91} C_VEL
LIN {X 0,Y 174.1,Z 1106.619,A -85,B 0,C 180,E1 31113.14,E2 31113.14} C_VEL
LIN {X 0,Y 200.392,Z 1088.876,A -85,B 0,C 180,E1 31119.284,E2 31119.284} C_VEL
LIN {X 0,Y 210.73,Z 1080.239,A -85,B 0,C 180,E1 31122.419,E2 31122.419} C_VEL
LIN {X 0,Y 221.22,Z 1070.957,A -85,B 0,C 180,E1 31125.218,E2 31125.218} C_VEL
LIN {X 0,Y 252.756,Z 1041.486,A -85,B 0,C 180,E1 31129.01,E2 31129.01} C_VEL
LIN {X 0,Y 262.961,Z 1030.344,A -85,B 0,C 180,E1 31130.034,E2 31130.034} C_VEL
LIN {X 0,Y 264.945,Z 1026.204,A -85,B 0,C 180,E1 31133.421,E2 31133.421} C_VEL
LIN {X 0,Y 266.286,Z 1023.788,A -85,B 0,C 180,E1 31136.726,E2 31136.726} C_VEL
LIN {X 0,Y 266.494,Z 1023.602,A -85,B 0,C 180,E1 31139.988,E2 31139.988} C_VEL
LIN {X 0,Y 263.969,Z 1028.809,A -85,B 0,C 180,E1 31145.752,E2 31145.752} C_VEL
LIN {X 0,Y 263.471,Z 1029.953,A -85,B 0,C 180,E1 31146.591,E2 31146.591} C_VEL
LIN {X 0,Y 233.92,Z 1060.594,A -85,B 0,C 180,E1 31149.988,E2 31149.988} C_VEL
LIN {X 0,Y 201.807,Z 1087.408,A -85,B 0,C 180,E1 31154.684,E2 31154.684} C_VEL
LIN {X 0,Y 167.043,Z 1110.871,A -85,B 0,C 180,E1 31162.259,E2 31162.259} C_VEL
LIN {X 0,Y 135.007,Z 1128.601,A -85,B 0,C 180,E1 31174.102,E2 31174.102} C_VEL
LIN {X 0,Y 110.682,Z 1140.339,A -85,B 0,C 180,E1 31191.966,E2 31191.966} C_VEL
LIN {X 0,Y 99.93,Z 1145.927,A -85,B 0,C 180,E1 31212.34,E2 31212.34} C_VEL
LIN {X 0,Y 98.685,Z 1147.36,A -85,B 0,C 180,E1 31229.992,E2 31229.992} C_VEL
LIN {X 0,Y 99.895,Z 1145.949,A -85,B 0,C 180,E1 31247.651,E2 31247.651} C_VEL
LIN {X 0,Y 110.686,Z 1140.408,A -85,B 0,C 180,E1 31268.016,E2 31268.016} C_VEL
LIN {X 0,Y 134.914,Z 1128.751,A -85,B 0,C 180,E1 31285.871,E2 31285.871} C_VEL
LIN {X 0,Y 166.931,Z 1111.06,A -85,B 0,C 180,E1 31297.736,E2 31297.736} C_VEL
LIN {X 0,Y 201.741,Z 1087.656,A -85,B 0,C 180,E1 31305.308,E2 31305.308} C_VEL
LIN {X 0,Y 235.467,Z 1059.46,A -85,B 0,C 180,E1 31310.195,E2 31310.195} C_VEL
LIN {X 0,Y 263.642,Z 1030.138,A -85,B 0,C 180,E1 31313.413,E2 31313.413} C_VEL
LIN {X 0,Y 265.885,Z 1025.059,A -85,B 0,C 180,E1 31318.38,E2 31318.38} C_VEL
LIN {X 0,Y 266.598,Z 1023.892,A -85,B 0,C 180,E1 31320.012,E2 31320.012} C_VEL
LIN {X 0,Y 266.341,Z 1024.143,A -85,B 0,C 180,E1 31323.273,E2 31323.273} C_VEL
LIN {X 0,Y 263.808,Z 1029.382,A -85,B 0,C 180,E1 31329.293,E2 31329.293} C_VEL
LIN {X 0,Y 262.65,Z 1031.083,A -85,B 0,C 180,E1 31329.906,E2 31329.906} C_VEL
LIN {X 0,Y 231.392,Z 1062.455,A -85,B 0,C 180,E1 31333.343,E2 31333.343} C_VEL
LIN {X 0,Y 198.87,Z 1088.485,A -85,B 0,C 180,E1 31338.272,E2 31338.272} C_VEL
LIN {X 0,Y 167.425,Z 1108.831,A -85,B 0,C 180,E1 31345.19,E2 31345.19} C_VEL
LIN {X 0,Y 136.505,Z 1125.224,A -85,B 0,C 180,E1 31356.426,E2 31356.426} C_VEL
LIN {X 0,Y 110.753,Z 1136.734,A -85,B 0,C 180,E1 31375.212,E2 31375.212} C_VEL
LIN {X 0,Y 100.908,Z 1140.94,A -85,B 0,C 180,E1 31392.532,E2 31392.532} C_VEL
LIN {X 0,Y 98.932,Z 1142.177,A -85,B 0,C 180,E1 31410.008,E2 31410.008} C_VEL
LIN {X 0,Y 100.96,Z 1140.906,A -85,B 0,C 180,E1 31427.475,E2 31427.475} C_VEL
LIN {X 0,Y 113.255,Z 1135.526,A -85,B 0,C 180,E1 31447.445,E2 31447.445} C_VEL
LIN {X 0,Y 139.177,Z 1123.761,A -85,B 0,C 180,E1 31464.745,E2 31464.745} C_VEL
LIN {X 0,Y 170.449,Z 1106.946,A -85,B 0,C 180,E1 31475.508,E2 31475.508} C_VEL
LIN {X 0,Y 205.803,Z 1083.251,A -85,B 0,C 180,E1 31482.858,E2 31482.858} C_VEL
LIN {X 0,Y 221.22,Z 1070.957,A -85,B 0,C 180,E1 31485.218,E2 31485.218} C_VEL
LIN {X 0,Y 231.88,Z 1061.074,A -85,B 0,C 180,E1 31487.71,E2 31487.71} C_VEL
LIN {X 0,Y 242.511,Z 1050.561,A -85,B 0,C 180,E1 31489.91,E2 31489.91} C_VEL
LIN {X 0,Y 257.524,Z 1035.228,A -85,B 0,C 180,E1 31491.375,E2 31491.375} C_VEL
LIN {X 0,Y 259.076,Z 1033.108,A -85,B 0,C 180,E1 31492.483,E2 31492.483} C_VEL
LIN {X 0,Y 260.889,Z 1029.79,A -85,B 0,C 180,E1 31496.658,E2 31496.658} C_VEL
LIN {X 0,Y 261.14,Z 1029.547,A -85,B 0,C 180,E1 31499.988,E2 31499.988} C_VEL
LIN {X 0,Y 258.688,Z 1034.279,A -85,B 0,C 180,E1 31505.28,E2 31505.28} C_VEL
LIN {X 0,Y 226.157,Z 1066.226,A -85,B 0,C 180,E1 31508.792,E2 31508.792} C_VEL
LIN {X 0,Y 190.182,Z 1094.098,A -85,B 0,C 180,E1 31514.063,E2 31514.063} C_VEL
LIN {X 0,Y 155.267,Z 1115.626,A -85,B 0,C 180,E1 31522.007,E2 31522.007} C_VEL
LIN {X 0,Y 124.017,Z 1131.395,A -85,B 0,C 180,E1 31534.434,E2 31534.434} C_VEL
LIN {X 0,Y 101.081,Z 1141.588,A -85,B 0,C 180,E1 31553.151,E2 31553.151} C_VEL
LIN {X 0,Y 92.308,Z 1145.716,A -85,B 0,C 180,E1 31570.827,E2 31570.827} C_VEL
LIN {X 0,Y 90.759,Z 1147.152,A -85,B 0,C 180,E1 31589.992,E2 31589.992} C_VEL
LIN {X 0,Y 92.276,Z 1145.739,A -85,B 0,C 180,E1 31609.163,E2 31609.163} C_VEL
LIN {X 0,Y 104.401,Z 1140.194,A -85,B 0,C 180,E1 31630.765,E2 31630.765} C_VEL
LIN {X 0,Y 130.489,Z 1128.533,A -85,B 0,C 180,E1 31648.853,E2 31648.853} C_VEL
LIN {X 0,Y 166.064,Z 1109.627,A -85,B 0,C 180,E1 31660.908,E2 31660.908} C_VEL
LIN {X 0,Y 203.204,Z 1084.943,A -85,B 0,C 180,E1 31668.12,E2 31668.12} C_VEL
LIN {X 0,Y 238.423,Z 1055.355,A -85,B 0,C 180,E1 31672.616,E2 31672.616} C_VEL
LIN {X 0,Y 258.707,Z 1034.67,A -85,B 0,C 180,E1 31674.612,E2 31674.612} C_VEL
LIN {X 0,Y 261.219,Z 1029.862,A -85,B 0,C 180,E1 31680.012,E2 31680.012} C_VEL
LIN {X 0,Y 260.951,Z 1030.136,A -85,B 0,C 180,E1 31683.341,E2 31683.341} C_VEL
LIN {X 0,Y 258.381,Z 1034.673,A -85,B 0,C 180,E1 31688.457,E2 31688.457} C_VEL
LIN {X 0,Y 225.633,Z 1066.254,A -85,B 0,C 180,E1 31691.887,E2 31691.887} C_VEL
LIN {X 0,Y 190.237,Z 1093.075,A -85,B 0,C 180,E1 31697.122,E2 31697.122} C_VEL
LIN {X 0,Y 154.877,Z 1114.172,A -85,B 0,C 180,E1 31705.198,E2 31705.198} C_VEL
LIN {X 0,Y 123.607,Z 1129.054,A -85,B 0,C 180,E1 31717.828,E2 31717.828} C_VEL
LIN {X 0,Y 100.009,Z 1138.515,A -85,B 0,C 180,E1 31737.986,E2 31737.986} C_VEL
LIN {X 0,Y 91.277,Z 1142.083,A -85,B 0,C 180,E1 31760.453,E2 31760.453} C_VEL
LIN {X 0,Y 90.968,Z 1142.36,A -85,B 0,C 180,E1 31770.838,E2 31770.838} C_VEL
LIN {X 0,Y 93.403,Z 1141.115,A -85,B 0,C 180,E1 31788.94,E2 31788.94} C_VEL
LIN {X 0,Y 110.561,Z 1134.353,A -85,B 0,C 180,E1 31813.262,E2 31813.262} C_VEL
LIN {X 0,Y 140.271,Z 1121.355,A -85,B 0,C 180,E1 31829.794,E2 31829.794} C_VEL
LIN {X 0,Y 171.757,Z 1104.473,A -85,B 0,C 180,E1 31839.076,E2 31839.076} C_VEL
LIN {X 0,Y 205.588,Z 1081.951,A -85,B 0,C 180,E1 31845.321,E2 31845.321} C_VEL
LIN {X 0,Y 238.839,Z 1054.135,A -85,B 0,C 180,E1 31849.531,E2 31849.531} C_VEL
LIN {X 0,Y 242.511,Z 1050.561,A -85,B 0,C 180,E1 31849.91,E2 31849.91} C_VEL
LIN {X 0,Y 249.95,Z 1042.863,A -85,B 0,C 180,E1 31851.355,E2 31851.355} C_VEL
LIN {X 0,Y 253.746,Z 1038.153,A -85,B 0,C 180,E1 31853.331,E2 31853.331} C_VEL
LIN {X 0,Y 253.956,Z 1037.818,A -85,B 0,C 180,E1 31853.662,E2 31853.662} C_VEL
LIN {X 0,Y 255.378,Z 1035.688,A -85,B 0,C 180,E1 31856.586,E2 31856.586} C_VEL
LIN {X 0,Y 255.69,Z 1035.417,A -85,B 0,C 180,E1 31859.987,E2 31859.987} C_VEL
LIN {X 0,Y 253.224,Z 1039.133,A -85,B 0,C 180,E1 31864.001,E2 31864.001} C_VEL
LIN {X 0,Y 221.431,Z 1068.987,A -85,B 0,C 180,E1 31867.144,E2 31867.144} C_VEL
LIN {X 0,Y 185.935,Z 1095.472,A -85,B 0,C 180,E1 31872.058,E2 31872.058} C_VEL
LIN {X 0,Y 149.189,Z 1117.146,A -85,B 0,C 180,E1 31880.03,E2 31880.03} C_VEL
LIN {X 0,Y 114.34,Z 1133.511,A -85,B 0,C 180,E1 31894.073,E2 31894.073} C_VEL
LIN {X 0,Y 89.593,Z 1143.477,A -85,B 0,C 180,E1 31917.658,E2 31917.658} C_VEL
LIN {X 0,Y 82.794,Z 1146.565,A -85,B 0,C 180,E1 31939.446,E2 31939.446} C_VEL
LIN {X 0,Y 82.829,Z 1146.944,A -85,B 0,C 180,E1 31949.991,E2 31949.991} C_VEL
LIN {X 0,Y 84.73,Z 1145.528,A -85,B 0,C 180,E1 31970.946,E2 31970.946} C_VEL
LIN {X 0,Y 98.394,Z 1139.981,A -85,B 0,C 180,E1 31993.853,E2 31993.853} C_VEL
LIN {X 0,Y 124.928,Z 1128.987,A -85,B 0,C 180,E1 32011.351,E2 32011.351} C_VEL
LIN {X 0,Y 158.852,Z 1112.017,A -85,B 0,C 180,E1 32022.504,E2 32022.504} C_VEL
LIN {X 0,Y 192.935,Z 1090.876,A -85,B 0,C 180,E1 32029.084,E2 32029.084} C_VEL
LIN {X 0,Y 226.848,Z 1064.669,A -85,B 0,C 180,E1 32033.45,E2 32033.45} C_VEL
LIN {X 0,Y 253.885,Z 1038.745,A -85,B 0,C 180,E1 32036.164,E2 32036.164} C_VEL
LIN {X 0,Y 255.733,Z 1035.741,A -85,B 0,C 180,E1 32040.013,E2 32040.013} C_VEL
LIN {X 0,Y 255.43,Z 1036.013,A -85,B 0,C 180,E1 32043.413,E2 32043.413} C_VEL
LIN {X 0,Y 253.846,Z 1038.513,A -85,B 0,C 180,E1 32046.868,E2 32046.868} C_VEL
LIN {X 0,Y 222.421,Z 1067.861,A -85,B 0,C 180,E1 32050.075,E2 32050.075} C_VEL
LIN {X 0,Y 188.029,Z 1093.295,A -85,B 0,C 180,E1 32054.781,E2 32054.781} C_VEL
LIN {X 0,Y 151.627,Z 1114.387,A -85,B 0,C 180,E1 32062.447,E2 32062.447} C_VEL
LIN {X 0,Y 118.842,Z 1129.265,A -85,B 0,C 180,E1 32074.763,E2 32074.763} C_VEL
LIN {X 0,Y 95.76,Z 1137.876,A -85,B 0,C 180,E1 32092.339,E2 32092.339} C_VEL
LIN {X 0,Y 83.453,Z 1142.291,A -85,B 0,C 180,E1 32119.549,E2 32119.549} C_VEL
LIN {X 0,Y 83.142,Z 1142.591,A -85,B 0,C 180,E1 32130.009,E2 32130.009} C_VEL
LIN {X 0,Y 85.899,Z 1141.324,A -85,B 0,C 180,E1 32150.667,E2 32150.667} C_VEL
LIN {X 0,Y 104.863,Z 1134.564,A -85,B 0,C 180,E1 32176.267,E2 32176.267} C_VEL
LIN {X 0,Y 136.4,Z 1121.571,A -85,B 0,C 180,E1 32192.717,E2 32192.717} C_VEL
LIN {X 0,Y 170.385,Z 1103.925,A -85,B 0,C 180,E1 32201.894,E2 32201.894} C_VEL
LIN {X 0,Y 203.707,Z 1082.185,A -85,B 0,C 180,E1 32207.5,E2 32207.5} C_VEL
LIN {X 0,Y 237.52,Z 1054.39,A -85,B 0,C 180,E1 32211.422,E2 32211.422} C_VEL
LIN {X 0,Y 252.677,Z 1039.434,A -85,B 0,C 180,E1 32212.813,E2 32212.813} C_VEL
LIN {X 0,Y 253.956,Z 1037.818,A -85,B 0,C 180,E1 32213.662,E2 32213.662} C_VEL
LIN {X 0,Y 253.361,Z 1037.729,A -85,B 0,C 180,E1 32216.618,E2 32216.618} C_VEL
LIN {X 0,Y 249.239,Z 1042.283,A -85,B 0,C 180,E1 32221.581,E2 32221.581} C_VEL
LIN {X 0,Y 248.756,Z 1043.038,A -85,B 0,C 180,E1 32222.465,E2 32222.465} C_VEL
LIN {X 0,Y 215.065,Z 1073.177,A -85,B 0,C 180,E1 32225.625,E2 32225.625} C_VEL
LIN {X 0,Y 180.865,Z 1097.453,A -85,B 0,C 180,E1 32230.133,E2 32230.133} C_VEL
LIN {X 0,Y 146.59,Z 1116.926,A -85,B 0,C 180,E1 32237.026,E2 32237.026} C_VEL
LIN {X 0,Y 109.959,Z 1133.294,A -85,B 0,C 180,E1 32250.534,E2 32250.534} C_VEL
LIN {X 0,Y 85.018,Z 1142.422,A -85,B 0,C 180,E1 32271.398,E2 32271.398} C_VEL
LIN {X 0,Y 74.982,Z 1146.357,A -85,B 0,C 180,E1 32298.332,E2 32298.332} C_VEL
LIN {X 0,Y 74.905,Z 1146.736,A -85,B 0,C 180,E1 32309.99,E2 32309.99} C_VEL
LIN {X 0,Y 77.291,Z 1145.318,A -85,B 0,C 180,E1 32333.072,E2 32333.072} C_VEL
LIN {X 0,Y 92.702,Z 1139.768,A -85,B 0,C 180,E1 32357.337,E2 32357.337} C_VEL
LIN {X 0,Y 121.371,Z 1128.709,A -85,B 0,C 180,E1 32374.818,E2 32374.818} C_VEL
LIN {X 0,Y 160.156,Z 1109.922,A -85,B 0,C 180,E1 32386.144,E2 32386.144} C_VEL
LIN {X 0,Y 198.676,Z 1085.8,A -85,B 0,C 180,E1 32392.459,E2 32392.459} C_VEL
LIN {X 0,Y 236.376,Z 1055.334,A -85,B 0,C 180,E1 32396.462,E2 32396.462} C_VEL
LIN {X 0,Y 248.869,Z 1043.282,A -85,B 0,C 180,E1 32397.534,E2 32397.534} C_VEL
LIN {X 0,Y 250.079,Z 1041.471,A -85,B 0,C 180,E1 32400.013,E2 32400.013} C_VEL
LIN {X 0,Y 249.232,Z 1042.507,A -85,B 0,C 180,E1 32404.66,E2 32404.66} C_VEL
LIN {X 0,Y 248.446,Z 1043.532,A -85,B 0,C 180,E1 32405.569,E2 32405.569} C_VEL
LIN {X 0,Y 212.789,Z 1074.792,A -85,B 0,C 180,E1 32408.921,E2 32408.921} C_VEL
LIN {X 0,Y 173.986,Z 1100.996,A -85,B 0,C 180,E1 32414.362,E2 32414.362} C_VEL
LIN {X 0,Y 135.744,Z 1120.7,A -85,B 0,C 180,E1 32423.176,E2 32423.176} C_VEL
LIN {X 0,Y 104.327,Z 1133.16,A -85,B 0,C 180,E1 32436.999,E2 32436.999} C_VEL
LIN {X 0,Y 83.569,Z 1139.989,A -85,B 0,C 180,E1 32457.06,E2 32457.06} C_VEL
LIN {X 0,Y 75.662,Z 1142.499,A -85,B 0,C 180,E1 32478.458,E2 32478.458} C_VEL
LIN {X 0,Y 75.227,Z 1142.799,A -85,B 0,C 180,E1 32490.01,E2 32490.01} C_VEL
LIN {X 0,Y 78.499,Z 1141.533,A -85,B 0,C 180,E1 32512.718,E2 32512.718} C_VEL
LIN {X 0,Y 99.471,Z 1134.777,A -85,B 0,C 180,E1 32539.618,E2 32539.618} C_VEL
LIN {X 0,Y 129.823,Z 1123.097,A -85,B 0,C 180,E1 32554.77,E2 32554.77} C_VEL
LIN {X 0,Y 162.256,Z 1107.433,A -85,B 0,C 180,E1 32563.368,E2 32563.368} C_VEL
LIN {X 0,Y 200.344,Z 1083.73,A -85,B 0,C 180,E1 32569.491,E2 32569.491} C_VEL
LIN {X 0,Y 236.465,Z 1054.645,A -85,B 0,C 180,E1 32573.327,E2 32573.327} C_VEL
LIN {X 0,Y 248.411,Z 1043.202,A -85,B 0,C 180,E1 32574.363,E2 32574.363} C_VEL
LIN {X 0,Y 249.698,Z 1041.455,A -85,B 0,C 180,E1 32576.508,E2 32576.508} C_VEL
LIN {X 0,Y 250.057,Z 1041.127,A -85,B 0,C 180,E1 32579.987,E2 32579.987} C_VEL
LIN {X 0,Y 249.239,Z 1042.283,A -85,B 0,C 180,E1 32581.581,E2 32581.581} C_VEL
LIN {X 0,Y 246.057,Z 1045.657,A -85,B 0,C 180,E1 32582.274,E2 32582.274} C_VEL
LIN {X 0,Y 231.904,Z 1058.393,A -85,B 0,C 180,E1 32581.884,E2 32581.884} C_VEL
LIN {X 0,Y 195.966,Z 1086.561,A -85,B 0,C 180,E1 32585.42,E2 32585.42} C_VEL
LIN {X 0,Y 158.477,Z 1109.504,A -85,B 0,C 180,E1 32591.002,E2 32591.002} C_VEL
LIN {X 0,Y 118.164,Z 1128.386,A -85,B 0,C 180,E1 32601.605,E2 32601.605} C_VEL
LIN {X 0,Y 87.395,Z 1139.48,A -85,B 0,C 180,E1 32618.711,E2 32618.711} C_VEL
LIN {X 0,Y 69.982,Z 1145.084,A -85,B 0,C 180,E1 32644.329,E2 32644.329} C_VEL
LIN {X 0,Y 66.97,Z 1146.528,A -85,B 0,C 180,E1 32669.989,E2 32669.989} C_VEL
LIN {X 0,Y 69.962,Z 1145.108,A -85,B 0,C 180,E1 32695.655,E2 32695.655} C_VEL
LIN {X 0,Y 87.398,Z 1139.554,A -85,B 0,C 180,E1 32721.259,E2 32721.259} C_VEL
LIN {X 0,Y 121.28,Z 1127.179,A -85,B 0,C 180,E1 32739.533,E2 32739.533} C_VEL
LIN {X 0,Y 159.833,Z 1108.901,A -85,B 0,C 180,E1 32749.271,E2 32749.271} C_VEL
LIN {X 0,Y 197.775,Z 1085.572,A -85,B 0,C 180,E1 32754.79,E2 32754.79} C_VEL
LIN {X 0,Y 234.307,Z 1056.624,A -85,B 0,C 180,E1 32758.292,E2 32758.292} C_VEL
LIN {X 0,Y 242.456,Z 1049.015,A -85,B 0,C 180,E1 32758.916,E2 32758.916} C_VEL
LIN {X 0,Y 244.321,Z 1047.102,A -85,B 0,C 180,E1 32760.013,E2 32760.013} C_VEL
LIN {X 0,Y 243.957,Z 1047.404,A -85,B 0,C 180,E1 32763.574,E2 32763.574} C_VEL
LIN {X 0,Y 243.03,Z 1048.329,A -85,B 0,C 180,E1 32764.085,E2 32764.085} C_VEL
LIN {X 0,Y 209.868,Z 1076.383,A -85,B 0,C 180,E1 32766.961,E2 32766.961} C_VEL
LIN {X 0,Y 172.162,Z 1101.215,A -85,B 0,C 180,E1 32771.759,E2 32771.759} C_VEL
LIN {X 0,Y 132.254,Z 1121.124,A -85,B 0,C 180,E1 32780.126,E2 32780.126} C_VEL
LIN {X 0,Y 99.696,Z 1133.371,A -85,B 0,C 180,E1 32793.306,E2 32793.306} C_VEL
LIN {X 0,Y 76.967,Z 1140.199,A -85,B 0,C 180,E1 32813.814,E2 32813.814} C_VEL
LIN {X 0,Y 67.894,Z 1142.707,A -85,B 0,C 180,E1 32837.116,E2 32837.116} C_VEL
LIN {X 0,Y 67.311,Z 1143.007,A -85,B 0,C 180,E1 32850.011,E2 32850.011} C_VEL
LIN {X 0,Y 71.207,Z 1141.742,A -85,B 0,C 180,E1 32875.198,E2 32875.198} C_VEL
LIN {X 0,Y 94.456,Z 1134.989,A -85,B 0,C 180,E1 32903.339,E2 32903.339} C_VEL
LIN {X 0,Y 126.598,Z 1123.314,A -85,B 0,C 180,E1 32918.071,E2 32918.071} C_VEL
LIN {X 0,Y 160.14,Z 1107.655,A -85,B 0,C 180,E1 32926.125,E2 32926.125} C_VEL
LIN {X 0,Y 199.037,Z 1083.965,A -85,B 0,C 180,E1 32931.765,E2 32931.765} C_VEL
LIN {X 0,Y 235.673,Z 1054.899,A -85,B 0,C 180,E1 32935.248,E2 32935.248} C_VEL
LIN {X 0,Y 243.082,Z 1047.946,A -85,B 0,C 180,E1 32935.83,E2 32935.83} C_VEL
LIN {X 0,Y 243.908,Z 1047.104,A -85,B 0,C 180,E1 32936.425,E2 32936.425} C_VEL
LIN {X 0,Y 244.305,Z 1046.781,A -85,B 0,C 180,E1 32939.987,E2 32939.987} C_VEL
LIN {X 0,Y 242.48,Z 1048.655,A -85,B 0,C 180,E1 32941.057,E2 32941.057} C_VEL
LIN {X 0,Y 231.904,Z 1058.393,A -85,B 0,C 180,E1 32941.884,E2 32941.884} C_VEL
LIN {X 0,Y 218.308,Z 1069.574,A -85,B 0,C 180,E1 32941.976,E2 32941.976} C_VEL
LIN {X 0,Y 204.3,Z 1080.001,A -85,B 0,C 180,E1 32942.166,E2 32942.166} C_VEL
LIN {X 0,Y 167.734,Z 1103.46,A -85,B 0,C 180,E1 32946.424,E2 32946.424} C_VEL
LIN {X 0,Y 128.139,Z 1122.978,A -85,B 0,C 180,E1 32954.058,E2 32954.058} C_VEL
LIN {X 0,Y 93.59,Z 1135.843,A -85,B 0,C 180,E1 32967.057,E2 32967.057} C_VEL
LIN {X 0,Y 69.057,Z 1143.141,A -85,B 0,C 180,E1 32988.821,E2 32988.821} C_VEL
LIN {X 0,Y 59.433,Z 1145.938,A -85,B 0,C 180,E1 33015.217,E2 33015.217} C_VEL
LIN {X 0,Y 59.048,Z 1146.32,A -85,B 0,C 180,E1 33029.987,E2 33029.987} C_VEL
LIN {X 0,Y 62.838,Z 1144.898,A -85,B 0,C 180,E1 33058.818,E2 33058.818} C_VEL
LIN {X 0,Y 85.764,Z 1138.358,A -85,B 0,C 180,E1 33088.042,E2 33088.042} C_VEL
LIN {X 0,Y 118.666,Z 1126.962,A -85,B 0,C 180,E1 33103.238,E2 33103.238} C_VEL
LIN {X 0,Y 156.893,Z 1109.562,A -85,B 0,C 180,E1 33111.909,E2 33111.909} C_VEL
LIN {X 0,Y 197.202,Z 1085.342,A -85,B 0,C 180,E1 33117.145,E2 33117.145} C_VEL
LIN {X 0,Y 233.957,Z 1056.593,A -85,B 0,C 180,E1 33120.255,E2 33120.255} C_VEL
LIN {X 0,Y 238.37,Z 1052.536,A -85,B 0,C 180,E1 33120.735,E2 33120.735} C_VEL
LIN {X 0,Y 237.642,Z 1053.175,A -85,B 0,C 180,E1 33122.544,E2 33122.544} C_VEL
LIN {X 0,Y 203.508,Z 1080.55,A -85,B 0,C 180,E1 33125.296,E2 33125.296} C_VEL
LIN {X 0,Y 168.909,Z 1102.393,A -85,B 0,C 180,E1 33129.373,E2 33129.373} C_VEL
LIN {X 0,Y 129.705,Z 1121.336,A -85,B 0,C 180,E1 33136.785,E2 33136.785} C_VEL
LIN {X 0,Y 94.716,Z 1133.842,A -85,B 0,C 180,E1 33149.692,E2 33149.692} C_VEL
LIN {X 0,Y 70.665,Z 1140.408,A -85,B 0,C 180,E1 33169.98,E2 33169.98} C_VEL
LIN {X 0,Y 60.172,Z 1142.915,A -85,B 0,C 180,E1 33195.429,E2 33195.429} C_VEL
LIN {X 0,Y 59.413,Z 1143.214,A -85,B 0,C 180,E1 33210.013,E2 33210.013} C_VEL
LIN {X 0,Y 64.075,Z 1141.951,A -85,B 0,C 180,E1 33238.238,E2 33238.238} C_VEL
LIN {X 0,Y 89.884,Z 1135.201,A -85,B 0,C 180,E1 33267.457,E2 33267.457} C_VEL
LIN {X 0,Y 123.82,Z 1123.529,A -85,B 0,C 180,E1 33281.524,E2 33281.524} C_VEL
LIN {X 0,Y 160.05,Z 1106.989,A -85,B 0,C 180,E1 33289.21,E2 33289.21} C_VEL
LIN {X 0,Y 198.047,Z 1084.199,A -85,B 0,C 180,E1 33294.06,E2 33294.06} C_VEL
LIN {X 0,Y 234.409,Z 1055.818,A -85,B 0,C 180,E1 33297.136,E2 33297.136} C_VEL
LIN {X 0,Y 237.553,Z 1052.917,A -85,B 0,C 180,E1 33297.362,E2 33297.362} C_VEL
LIN {X 0,Y 238.36,Z 1052.205,A -85,B 0,C 180,E1 33299.243,E2 33299.243} C_VEL
LIN {X 0,Y 204.3,Z 1080.001,A -85,B 0,C 180,E1 33302.166,E2 33302.166} C_VEL
LIN {X 0,Y 189.74,Z 1089.773,A -85,B 0,C 180,E1 33302.424,E2 33302.424} C_VEL
LIN {X 0,Y 174.77,Z 1098.79,A -85,B 0,C 180,E1 33302.733,E2 33302.733} C_VEL
LIN {X 0,Y 137.76,Z 1117.836,A -85,B 0,C 180,E1 33308.124,E2 33308.124} C_VEL
LIN {X 0,Y 99.827,Z 1132.628,A -85,B 0,C 180,E1 33318.294,E2 33318.294} C_VEL
LIN {X 0,Y 67.72,Z 1141.783,A -85,B 0,C 180,E1 33338.439,E2 33338.439} C_VEL
LIN {X 0,Y 51.741,Z 1145.729,A -85,B 0,C 180,E1 33372.957,E2 33372.957} C_VEL
LIN {X 0,Y 51.108,Z 1146.112,A -85,B 0,C 180,E1 33389.985,E2 33389.985} C_VEL
LIN {X 0,Y 59.418,Z 1143.819,A -85,B 0,C 180,E1 33430.184,E2 33430.184} C_VEL
LIN {X 0,Y 90.169,Z 1135.721,A -85,B 0,C 180,E1 33457.526,E2 33457.526} C_VEL
LIN {X 0,Y 129.532,Z 1121.586,A -85,B 0,C 180,E1 33470.207,E2 33470.207} C_VEL
LIN {X 0,Y 169.777,Z 1101.932,A -85,B 0,C 180,E1 33476.687,E2 33476.687} C_VEL
LIN {X 0,Y 210.226,Z 1075.698,A -85,B 0,C 180,E1 33480.578,E2 33480.578} C_VEL
LIN {X 0,Y 221.66,Z 1066.828,A -85,B 0,C 180,E1 33481.638,E2 33481.638} C_VEL
LIN {X 0,Y 185.32,Z 1092.439,A -85,B 0,C 180,E1 33484.707,E2 33484.707} C_VEL
LIN {X 0,Y 146.048,Z 1113.548,A -85,B 0,C 180,E1 33489.777,E2 33489.777} C_VEL
LIN {X 0,Y 107.917,Z 1128.741,A -85,B 0,C 180,E1 33498.634,E2 33498.634} C_VEL
LIN {X 0,Y 74.474,Z 1138.393,A -85,B 0,C 180,E1 33515.549,E2 33515.549} C_VEL
LIN {X 0,Y 52.514,Z 1143.124,A -85,B 0,C 180,E1 33553.245,E2 33553.245} C_VEL
LIN {X 0,Y 51.494,Z 1143.421,A -85,B 0,C 180,E1 33570.015,E2 33570.015} C_VEL
LIN {X 0,Y 57.167,Z 1142.16,A -85,B 0,C 180,E1 33602.026,E2 33602.026} C_VEL
LIN {X 0,Y 80.026,Z 1136.933,A -85,B 0,C 180,E1 33628.448,E2 33628.448} C_VEL
LIN {X 0,Y 114.648,Z 1126.371,A -85,B 0,C 180,E1 33643.31,E2 33643.31} C_VEL
LIN {X 0,Y 157.086,Z 1108.088,A -85,B 0,C 180,E1 33651.826,E2 33651.826} C_VEL
LIN {X 0,Y 197.379,Z 1084.433,A -85,B 0,C 180,E1 33656.373,E2 33656.373} C_VEL
LIN {X 0,Y 222.466,Z 1065.904,A -85,B 0,C 180,E1 33658.334,E2 33658.334} C_VEL
LIN {X 0,Y 183.811,Z 1093.415,A -85,B 0,C 180,E1 33661.743,E2 33661.743} C_VEL
LIN {X 0,Y 174.77,Z 1098.79,A -85,B 0,C 180,E1 33662.733,E2 33662.733} C_VEL
LIN {X 0,Y 159.35,Z 1107.086,A -85,B 0,C 180,E1 33663.158,E2 33663.158} C_VEL
LIN {X 0,Y 143.599,Z 1114.596,A -85,B 0,C 180,E1 33663.725,E2 33663.725} C_VEL
LIN {X 0,Y 104.499,Z 1130.073,A -85,B 0,C 180,E1 33671.62,E2 33671.62} C_VEL
LIN {X 0,Y 68.608,Z 1140.307,A -85,B 0,C 180,E1 33687.924,E2 33687.924} C_VEL
LIN {X 0,Y 49.365,Z 1144.452,A -85,B 0,C 180,E1 33712.112,E2 33712.112} C_VEL
LIN {X 0,Y 43.181,Z 1145.904,A -85,B 0,C 180,E1 33749.983,E2 33749.983} C_VEL
LIN {X 0,Y 49.35,Z 1144.477,A -85,B 0,C 180,E1 33787.864,E2 33787.864} C_VEL
LIN {X 0,Y 74.713,Z 1138.883,A -85,B 0,C 180,E1 33816.122,E2 33816.122} C_VEL
LIN {X 0,Y 111.457,Z 1127.851,A -85,B 0,C 180,E1 33830.215,E2 33830.215} C_VEL
LIN {X 0,Y 155.397,Z 1109.14,A -85,B 0,C 180,E1 33837.886,E2 33837.886} C_VEL
LIN {X 0,Y 188.36,Z 1090.454,A -85,B 0,C 180,E1 33841.207,E2 33841.207} C_VEL
LIN {X 0,Y 189.906,Z 1089.45,A -85,B 0,C 180,E1 33841.79,E2 33841.79} C_VEL
LIN {X 0,Y 151.391,Z 1110.733,A -85,B 0,C 180,E1 33845.765,E2 33845.765} C_VEL
LIN {X 0,Y 114.943,Z 1125.849,A -85,B 0,C 180,E1 33852.102,E2 33852.102} C_VEL
LIN {X 0,Y 76.085,Z 1137.231,A -85,B 0,C 180,E1 33866.368,E2 33866.368} C_VEL
LIN {X 0,Y 50.535,Z 1142.4,A -85,B 0,C 180,E1 33893.174,E2 33893.174} C_VEL
LIN {X 0,Y 43.591,Z 1143.629,A -85,B 0,C 180,E1 33930.017,E2 33930.017} C_VEL
LIN {X 0,Y 50.577,Z 1142.37,A -85,B 0,C 180,E1 33966.828,E2 33966.828} C_VEL
LIN {X 0,Y 82.361,Z 1135.623,A -85,B 0,C 180,E1 33996.924,E2 33996.924} C_VEL
LIN {X 0,Y 119.323,Z 1124.095,A -85,B 0,C 180,E1 34008.785,E2 34008.785} C_VEL
LIN {X 0,Y 155.976,Z 1108.399,A -85,B 0,C 180,E1 34014.731,E2 34014.731} C_VEL
LIN {X 0,Y 190.246,Z 1089.002,A -85,B 0,C 180,E1 34018.169,E2 34018.169} C_VEL
LIN {X 0,Y 188.618,Z 1090.06,A -85,B 0,C 180,E1 34018.78,E2 34018.78} C_VEL
LIN {X 0,Y 151.687,Z 1110.754,A -85,B 0,C 180,E1 34022.614,E2 34022.614} C_VEL
LIN {X 0,Y 143.599,Z 1114.596,A -85,B 0,C 180,E1 34023.725,E2 34023.725} C_VEL
LIN {X 0,Y 127.477,Z 1121.34,A -85,B 0,C 180,E1 34024.455,E2 34024.455} C_VEL
LIN {X 0,Y 111.118,Z 1127.25,A -85,B 0,C 180,E1 34025.443,E2 34025.443} C_VEL
LIN {X 0,Y 71.582,Z 1138.644,A -85,B 0,C 180,E1 34037.973,E2 34037.973} C_VEL
LIN {X 0,Y 43.279,Z 1144.24,A -85,B 0,C 180,E1 34065.534,E2 34065.534} C_VEL
LIN {X 0,Y 35.234,Z 1145.696,A -85,B 0,C 180,E1 34109.979,E2 34109.979} C_VEL
LIN {X 0,Y 45.1,Z 1143.979,A -85,B 0,C 180,E1 34157.887,E2 34157.887} C_VEL
LIN {X 0,Y 78.38,Z 1137.08,A -85,B 0,C 180,E1 34185.101,E2 34185.101} C_VEL
LIN {X 0,Y 117.725,Z 1124.943,A -85,B 0,C 180,E1 34195.822,E2 34195.822} C_VEL
LIN {X 0,Y 157.504,Z 1107.782,A -85,B 0,C 180,E1 34201.132,E2 34201.132} C_VEL
LIN {X 0,Y 160.398,Z 1106.279,A -85,B 0,C 180,E1 34201.395,E2 34201.395} C_VEL
LIN {X 0,Y 147.4,Z 1112.507,A -85,B 0,C 180,E1 34203.092,E2 34203.092} C_VEL
LIN {X 0,Y 107.483,Z 1128.041,A -85,B 0,C 180,E1 34209.373,E2 34209.373} C_VEL
LIN {X 0,Y 66.434,Z 1138.813,A -85,B 0,C 180,E1 34224.206,E2 34224.206} C_VEL
LIN {X 0,Y 37.581,Z 1143.54,A -85,B 0,C 180,E1 34266.245,E2 34266.245} C_VEL
LIN {X 0,Y 35.668,Z 1143.836,A -85,B 0,C 180,E1 34290.021,E2 34290.021} C_VEL
LIN {X 0,Y 44.441,Z 1142.579,A -85,B 0,C 180,E1 34333.013,E2 34333.013} C_VEL
LIN {X 0,Y 79.552,Z 1135.835,A -85,B 0,C 180,E1 34362.266,E2 34362.266} C_VEL
LIN {X 0,Y 117.891,Z 1124.356,A -85,B 0,C 180,E1 34372.589,E2 34372.589} C_VEL
LIN {X 0,Y 157.973,Z 1107.323,A -85,B 0,C 180,E1 34377.946,E2 34377.946} C_VEL
LIN {X 0,Y 160.596,Z 1105.993,A -85,B 0,C 180,E1 34378.592,E2 34378.592} C_VEL
LIN {X 0,Y 121.455,Z 1123.437,A -85,B 0,C 180,E1 34383.517,E2 34383.517} C_VEL
LIN {X 0,Y 111.118,Z 1127.25,A -85,B 0,C 180,E1 34385.443,E2 34385.443} C_VEL
LIN {X 0,Y 94.517,Z 1132.334,A -85,B 0,C 180,E1 34386.775,E2 34386.775} C_VEL
LIN {X 0,Y 77.694,Z 1136.538,A -85,B 0,C 180,E1 34388.629,E2 34388.629} C_VEL
LIN {X 0,Y 49.497,Z 1142.291,A -85,B 0,C 180,E1 34403.278,E2 34403.278} C_VEL
LIN {X 0,Y 29.649,Z 1145.1,A -85,B 0,C 180,E1 34439.238,E2 34439.238} C_VEL
LIN {X 0,Y 27.289,Z 1145.488,A -85,B 0,C 180,E1 34469.972,E2 34469.972} C_VEL
LIN {X 0,Y 37.933,Z 1144.056,A -85,B 0,C 180,E1 34522.988,E2 34522.988} C_VEL
LIN {X 0,Y 70.563,Z 1138.261,A -85,B 0,C 180,E1 34548.811,E2 34548.811} C_VEL
LIN {X 0,Y 112.585,Z 1126.472,A -85,B 0,C 180,E1 34559.089,E2 34559.089} C_VEL
LIN {X 0,Y 130.403,Z 1119.807,A -85,B 0,C 180,E1 34561.464,E2 34561.464} C_VEL
LIN {X 0,Y 91.799,Z 1132.548,A -85,B 0,C 180,E1 34568.04,E2 34568.04} C_VEL
LIN {X 0,Y 50.51,Z 1141.245,A -85,B 0,C 180,E1 34585.886,E2 34585.886} C_VEL
LIN {X 0,Y 30.466,Z 1143.748,A -85,B 0,C 180,E1 34620.205,E2 34620.205} C_VEL
LIN {X 0,Y 27.767,Z 1144.044,A -85,B 0,C 180,E1 34650.027,E2 34650.027} C_VEL
LIN {X 0,Y 38.984,Z 1142.788,A -85,B 0,C 180,E1 34701.048,E2 34701.048} C_VEL
LIN {X 0,Y 77.481,Z 1136.046,A -85,B 0,C 180,E1 34727.94,E2 34727.94} C_VEL
LIN {X 0,Y 115.713,Z 1125.07,A -85,B 0,C 180,E1 34736.284,E2 34736.284} C_VEL
LIN {X 0,Y 130.749,Z 1119.517,A -85,B 0,C 180,E1 34738.492,E2 34738.492} C_VEL
LIN {X 0,Y 91.263,Z 1132.996,A -85,B 0,C 180,E1 34744.946,E2 34744.946} C_VEL
LIN {X 0,Y 77.694,Z 1136.538,A -85,B 0,C 180,E1 34748.629,E2 34748.629} C_VEL
LIN {X 0,Y 60.842,Z 1139.994,A -85,B 0,C 180,E1 34751.443,E2 34751.443} C_VEL
LIN {X 0,Y 43.912,Z 1142.454,A -85,B 0,C 180,E1 34756.07,E2 34756.07} C_VEL
LIN {X 0,Y 23.126,Z 1144.889,A -85,B 0,C 180,E1 34789.024,E2 34789.024} C_VEL
LIN {X 0,Y 19.335,Z 1145.279,A -85,B 0,C 180,E1 34829.961,E2 34829.961} C_VEL
LIN {X 0,Y 33.693,Z 1143.844,A -85,B 0,C 180,E1 34894.027,E2 34894.027} C_VEL
LIN {X 0,Y 68.416,Z 1138.271,A -85,B 0,C 180,E1 34915.127,E2 34915.127} C_VEL
LIN {X 0,Y 98.962,Z 1130.594,A -85,B 0,C 180,E1 34921.483,E2 34921.483} C_VEL
LIN {X 0,Y 61.614,Z 1139.234,A -85,B 0,C 180,E1 34930.443,E2 34930.443} C_VEL
LIN {X 0,Y 34.484,Z 1143.026,A -85,B 0,C 180,E1 34948.554,E2 34948.554} C_VEL
LIN {X 0,Y 19.841,Z 1144.251,A -85,B 0,C 180,E1 35010.038,E2 35010.038} C_VEL
LIN {X 0,Y 41.442,Z 1142.165,A -85,B 0,C 180,E1 35078.473,E2 35078.473} C_VEL
LIN {X 0,Y 80.833,Z 1135.244,A -85,B 0,C 180,E1 35094.928,E2 35094.928} C_VEL
LIN {X 0,Y 99.307,Z 1130.377,A -85,B 0,C 180,E1 35098.496,E2 35098.496} C_VEL
LIN {X 0,Y 61.107,Z 1139.666,A -85,B 0,C 180,E1 35107.241,E2 35107.241} C_VEL
LIN {X 0,Y 43.912,Z 1142.454,A -85,B 0,C 180,E1 35116.07,E2 35116.07} C_VEL
LIN {X 0,Y 31.665,Z 1143.832,A -85,B 0,C 180,E1 35122.874,E2 35122.874} C_VEL
LIN {X 0,Y 12.732,Z 1144.883,A -85,B 0,C 180,E1 35155.168,E2 35155.168} C_VEL
LIN {X 0,Y 11.378,Z 1145.07,A -85,B 0,C 180,E1 35189.934,E2 35189.934} C_VEL
LIN {X 0,Y 31.016,Z 1143.633,A -85,B 0,C 180,E1 35267.577,E2 35267.577} C_VEL
LIN {X 0,Y 65.934,Z 1138.539,A -85,B 0,C 180,E1 35281.531,E2 35281.531} C_VEL
LIN {X 0,Y 31.465,Z 1143.235,A -85,B 0,C 180,E1 35295.704,E2 35295.704} C_VEL
LIN {X 0,Y 11.923,Z 1144.459,A -85,B 0,C 180,E1 35370.063,E2 35370.063} C_VEL
LIN {X 0,Y 31.498,Z 1143.207,A -85,B 0,C 180,E1 35444.258,E2 35444.258} C_VEL
LIN {X 0,Y 65.903,Z 1138.469,A -85,B 0,C 180,E1 35458.429,E2 35458.429} C_VEL
LIN {X 0,Y 31.041,Z 1143.606,A -85,B 0,C 180,E1 35472.404,E2 35472.404} C_VEL
LIN {X 0,Y 12.732,Z 1144.883,A -85,B 0,C 180,E1 35515.168,E2 35515.168} C_VEL
LIN {X 0,Y 8.338,Z 1144.976,A -85,B 0,C 180,E1 35557.684,E2 35557.684} C_VEL
LIN {X 0,Y 14.707,Z 1144.491,A -85,B 0,C 180,E1 35634.237,E2 35634.237} C_VEL
LIN {X 0,Y 23.17,Z 1143.942,A -85,B 0,C 180,E1 35640.14,E2 35640.14} C_VEL
LIN {X 0,Y 15.355,Z 1144.374,A -85,B 0,C 180,E1 35649.639,E2 35649.639} C_VEL
LIN {X 0,Y 3.994,Z 1144.667,A -85,B 0,C 180,E1 35730.189,E2 35730.189} C_VEL
LIN {X 0,Y 15.385,Z 1144.364,A -85,B 0,C 180,E1 35810.304,E2 35810.304} C_VEL
LIN {X 0,Y 23.191,Z 1143.915,A -85,B 0,C 180,E1 35819.86,E2 35819.86} C_VEL
LIN {X 0,Y 3.416,Z 1144.861,A -85,B 0,C 180,E1 35909.78,E2 35909.78} C_VEL
LIN {X 0,Y 14.707,Z 1144.491,A -85,B 0,C 180,E1 35994.237,E2 35994.237} C_VEL
LIN {X 0,Y 16.709,Z 1146.49,A -85,B 0,C 180,E1 35995.855,E2 35995.855} C_VEL
LIN {X 0,Y 16.709,Z 1164.5,A -85,B 0,C 180,E1 35995.855,E2 35995.855} C_VEL
LIN {X 0,Y 16.709,Z 1164.5,A -85,B 0,C 180,E1 35995.855,E2 35995.855}

